ABB RAPID module: 711802ba.mod

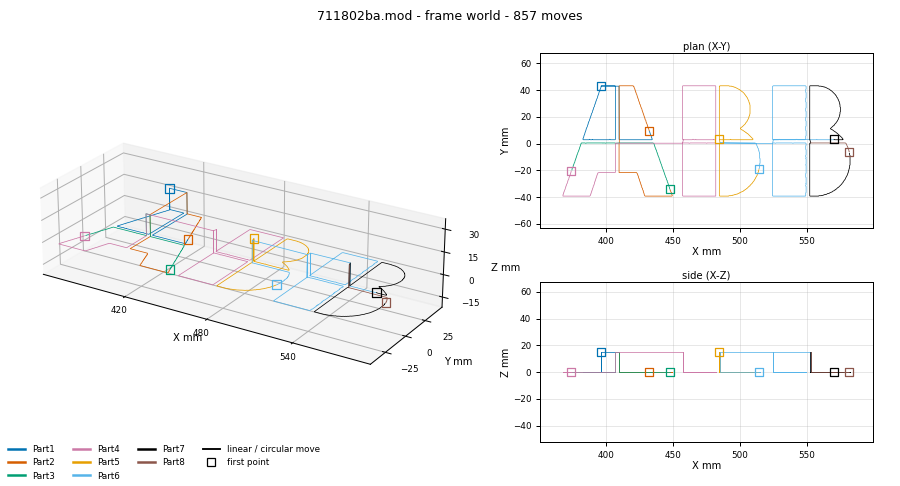
[picture p0: tool path of 711802ba.mod in frame world, 857 of 859 moves have a stored position in this frame; points joined in program order, loops and branches not executed]
MODULE ImageDraw
  ! Generated 2026-10-06 16:20 for ABB GoFa CRB 15000-5/0.95: 12 strokes
  PERS tooldata tPen:=[TRUE,[[0,0,120.0],[1,0,0,0]],[0.3,[0,0,60.0],[1,0,0,0],0,0,0]];
  PERS wobjdata wPaper:=[FALSE,TRUE,"",[[350,-90,0],[1,0,0,0]],[[0,0,0],[1,0,0,0]]];
  CONST robtarget pOrigin:=[[0,0,0],[0,1,0,0],[0,0,0,0],[9E9,9E9,9E9,9E9,9E9,9E9]];
  CONST jointtarget jHome:=[[0,0,0,0,30,0],[9E9,9E9,9E9,9E9,9E9,9E9]];
  CONST speeddata vDraw:=[40,100,5000,1000];
  CONST speeddata vApproach:=[20,100,5000,1000];
  CONST speeddata vTravel:=[200,200,5000,1000];

  PROC DrawImage()
    ConfL\Off;
    ConfJ\Off;
    MoveAbsJ jHome\NoEOffs,vTravel,fine,tPen;
    Part1;
    Part2;
    Part3;
    Part4;
    Part5;
    Part6;
    Part7;
    Part8;
    MoveAbsJ jHome\NoEOffs,vTravel,fine,tPen;
  ENDPROC

  PROC Part1()
    MoveL Offs(pOrigin,46.3,132.9,15.0),vTravel,z5,tPen\WObj:=wPaper;
    MoveL Offs(pOrigin,46.3,132.9,0.0),vApproach,fine,tPen\WObj:=wPaper;
    MoveL Offs(pOrigin,46.3,132.4,0.0),vDraw,z1,tPen\WObj:=wPaper;
    MoveL Offs(pOrigin,46.1,132.1,0.0),vDraw,z1,tPen\WObj:=wPaper;
    MoveL Offs(pOrigin,46.1,131.6,0.0),vDraw,z1,tPen\WObj:=wPaper;
    MoveL Offs(pOrigin,45.8,131.3,0.0),vDraw,z1,tPen\WObj:=wPaper;
    MoveL Offs(pOrigin,45.8,130.8,0.0),vDraw,z1,tPen\WObj:=wPaper;
    MoveL Offs(pOrigin,45.5,130.5,0.0),vDraw,z1,tPen\WObj:=wPaper;
    MoveL Offs(pOrigin,45.3,129.2,0.0),vDraw,z1,tPen\WObj:=wPaper;
    MoveL Offs(pOrigin,44.7,128.4,0.0),vDraw,z1,tPen\WObj:=wPaper;
    MoveL Offs(pOrigin,44.7,127.9,0.0),vDraw,z1,tPen\WObj:=wPaper;
    MoveL Offs(pOrigin,44.5,127.6,0.0),vDraw,z1,tPen\WObj:=wPaper;
    MoveL Offs(pOrigin,44.5,127.1,0.0),vDraw,z1,tPen\WObj:=wPaper;
    MoveL Offs(pOrigin,44.2,126.8,0.0),vDraw,z1,tPen\WObj:=wPaper;
    MoveL Offs(pOrigin,44.2,126.3,0.0),vDraw,z1,tPen\WObj:=wPaper;
    MoveL Offs(pOrigin,43.9,126.0,0.0),vDraw,z1,tPen\WObj:=wPaper;
    MoveL Offs(pOrigin,43.9,125.5,0.0),vDraw,z1,tPen\WObj:=wPaper;
    MoveL Offs(pOrigin,43.7,125.2,0.0),vDraw,z1,tPen\WObj:=wPaper;
    MoveL Offs(pOrigin,43.4,123.9,0.0),vDraw,z1,tPen\WObj:=wPaper;
    MoveL Offs(pOrigin,42.9,123.1,0.0),vDraw,z1,tPen\WObj:=wPaper;
    MoveL Offs(pOrigin,42.9,122.5,0.0),vDraw,z1,tPen\WObj:=wPaper;
    MoveL Offs(pOrigin,42.6,122.3,0.0),vDraw,z1,tPen\WObj:=wPaper;
    MoveL Offs(pOrigin,42.6,121.7,0.0),vDraw,z1,tPen\WObj:=wPaper;
    MoveL Offs(pOrigin,42.3,121.5,0.0),vDraw,z1,tPen\WObj:=wPaper;
    MoveL Offs(pOrigin,42.3,120.9,0.0),vDraw,z1,tPen\WObj:=wPaper;
    MoveL Offs(pOrigin,42.1,120.7,0.0),vDraw,z1,tPen\WObj:=wPaper;
    MoveL Offs(pOrigin,42.1,120.1,0.0),vDraw,z1,tPen\WObj:=wPaper;
    MoveL Offs(pOrigin,41.8,119.9,0.0),vDraw,z1,tPen\WObj:=wPaper;
    MoveL Offs(pOrigin,41.8,119.3,0.0),vDraw,z1,tPen\WObj:=wPaper;
    MoveL Offs(pOrigin,41.5,119.1,0.0),vDraw,z1,tPen\WObj:=wPaper;
    MoveL Offs(pOrigin,41.3,117.7,0.0),vDraw,z1,tPen\WObj:=wPaper;
    MoveL Offs(pOrigin,40.7,116.9,0.0),vDraw,z1,tPen\WObj:=wPaper;
    MoveL Offs(pOrigin,40.7,116.4,0.0),vDraw,z1,tPen\WObj:=wPaper;
    MoveL Offs(pOrigin,40.5,116.1,0.0),vDraw,z1,tPen\WObj:=wPaper;
    MoveL Offs(pOrigin,40.5,115.6,0.0),vDraw,z1,tPen\WObj:=wPaper;
    MoveL Offs(pOrigin,40.2,115.3,0.0),vDraw,z1,tPen\WObj:=wPaper;
    MoveL Offs(pOrigin,40.2,114.8,0.0),vDraw,z1,tPen\WObj:=wPaper;
    MoveL Offs(pOrigin,39.9,114.5,0.0),vDraw,z1,tPen\WObj:=wPaper;
    MoveL Offs(pOrigin,39.7,113.2,0.0),vDraw,z1,tPen\WObj:=wPaper;
    MoveL Offs(pOrigin,39.1,112.4,0.0),vDraw,z1,tPen\WObj:=wPaper;
    MoveL Offs(pOrigin,39.1,111.9,0.0),vDraw,z1,tPen\WObj:=wPaper;
    MoveL Offs(pOrigin,38.9,111.6,0.0),vDraw,z1,tPen\WObj:=wPaper;
    MoveL Offs(pOrigin,38.9,111.1,0.0),vDraw,z1,tPen\WObj:=wPaper;
    MoveL Offs(pOrigin,38.6,110.8,0.0),vDraw,z1,tPen\WObj:=wPaper;
    MoveL Offs(pOrigin,38.6,110.3,0.0),vDraw,z1,tPen\WObj:=wPaper;
    MoveL Offs(pOrigin,38.3,110.0,0.0),vDraw,z1,tPen\WObj:=wPaper;
    MoveL Offs(pOrigin,38.3,109.5,0.0),vDraw,z1,tPen\WObj:=wPaper;
    MoveL Offs(pOrigin,38.1,109.2,0.0),vDraw,z1,tPen\WObj:=wPaper;
    MoveL Offs(pOrigin,38.1,108.7,0.0),vDraw,z1,tPen\WObj:=wPaper;
    MoveL Offs(pOrigin,37.8,108.4,0.0),vDraw,z1,tPen\WObj:=wPaper;
    MoveL Offs(pOrigin,37.5,107.1,0.0),vDraw,z1,tPen\WObj:=wPaper;
    MoveL Offs(pOrigin,37.0,106.3,0.0),vDraw,z1,tPen\WObj:=wPaper;
    MoveL Offs(pOrigin,37.0,105.7,0.0),vDraw,z1,tPen\WObj:=wPaper;
    MoveL Offs(pOrigin,36.7,105.5,0.0),vDraw,z1,tPen\WObj:=wPaper;
    MoveL Offs(pOrigin,36.7,104.9,0.0),vDraw,z1,tPen\WObj:=wPaper;
    MoveL Offs(pOrigin,36.5,104.7,0.0),vDraw,z1,tPen\WObj:=wPaper;
    MoveL Offs(pOrigin,36.5,104.1,0.0),vDraw,z1,tPen\WObj:=wPaper;
    MoveL Offs(pOrigin,36.2,103.9,0.0),vDraw,z1,tPen\WObj:=wPaper;
    MoveL Offs(pOrigin,35.9,102.5,0.0),vDraw,z1,tPen\WObj:=wPaper;
    MoveL Offs(pOrigin,35.4,101.7,0.0),vDraw,z1,tPen\WObj:=wPaper;
    MoveL Offs(pOrigin,35.4,101.2,0.0),vDraw,z1,tPen\WObj:=wPaper;
    MoveL Offs(pOrigin,35.1,100.9,0.0),vDraw,z1,tPen\WObj:=wPaper;
    MoveL Offs(pOrigin,35.1,100.4,0.0),vDraw,z1,tPen\WObj:=wPaper;
    MoveL Offs(pOrigin,34.9,100.1,0.0),vDraw,z1,tPen\WObj:=wPaper;
    MoveL Offs(pOrigin,34.9,99.6,0.0),vDraw,z1,tPen\WObj:=wPaper;
    MoveL Offs(pOrigin,34.6,99.3,0.0),vDraw,z1,tPen\WObj:=wPaper;
    MoveL Offs(pOrigin,34.6,98.8,0.0),vDraw,z1,tPen\WObj:=wPaper;
    MoveL Offs(pOrigin,34.3,98.5,0.0),vDraw,z1,tPen\WObj:=wPaper;
    MoveL Offs(pOrigin,34.3,98.0,0.0),vDraw,z1,tPen\WObj:=wPaper;
    MoveL Offs(pOrigin,34.1,97.7,0.0),vDraw,z1,tPen\WObj:=wPaper;
    MoveL Offs(pOrigin,34.1,97.2,0.0),vDraw,z1,tPen\WObj:=wPaper;
    MoveL Offs(pOrigin,33.8,96.9,0.0),vDraw,z1,tPen\WObj:=wPaper;
    MoveL Offs(pOrigin,33.8,96.4,0.0),vDraw,z1,tPen\WObj:=wPaper;
    MoveL Offs(pOrigin,33.5,96.1,0.0),vDraw,z1,tPen\WObj:=wPaper;
    MoveL Offs(pOrigin,33.5,95.6,0.0),vDraw,z1,tPen\WObj:=wPaper;
    MoveL Offs(pOrigin,33.3,95.3,0.0),vDraw,z1,tPen\WObj:=wPaper;
    MoveL Offs(pOrigin,33.3,94.8,0.0),vDraw,z1,tPen\WObj:=wPaper;
    MoveL Offs(pOrigin,33.0,94.5,0.0),vDraw,z1,tPen\WObj:=wPaper;
    MoveL Offs(pOrigin,33.0,94.0,0.0),vDraw,z1,tPen\WObj:=wPaper;
    MoveL Offs(pOrigin,32.7,93.7,0.0),vDraw,z1,tPen\WObj:=wPaper;
    MoveL Offs(pOrigin,32.7,93.2,0.0),vDraw,z1,tPen\WObj:=wPaper;
    MoveL Offs(pOrigin,33.0,92.9,0.0),vDraw,z1,tPen\WObj:=wPaper;
    MoveL Offs(pOrigin,37.3,92.9,0.0),vDraw,z1,tPen\WObj:=wPaper;
    MoveL Offs(pOrigin,37.5,93.2,0.0),vDraw,z1,tPen\WObj:=wPaper;
    MoveL Offs(pOrigin,37.8,93.2,0.0),vDraw,z1,tPen\WObj:=wPaper;
    MoveL Offs(pOrigin,38.1,92.9,0.0),vDraw,z1,tPen\WObj:=wPaper;
    MoveL Offs(pOrigin,39.4,92.9,0.0),vDraw,z1,tPen\WObj:=wPaper;
    MoveL Offs(pOrigin,39.7,93.2,0.0),vDraw,z1,tPen\WObj:=wPaper;
    MoveL Offs(pOrigin,39.9,92.9,0.0),vDraw,z1,tPen\WObj:=wPaper;
    MoveL Offs(pOrigin,52.2,92.9,0.0),vDraw,z1,tPen\WObj:=wPaper;
    MoveL Offs(pOrigin,52.5,93.2,0.0),vDraw,z1,tPen\WObj:=wPaper;
    MoveL Offs(pOrigin,53.0,93.2,0.0),vDraw,z1,tPen\WObj:=wPaper;
    MoveL Offs(pOrigin,53.3,92.9,0.0),vDraw,z1,tPen\WObj:=wPaper;
    MoveL Offs(pOrigin,56.7,92.9,0.0),vDraw,z1,tPen\WObj:=wPaper;
    MoveL Offs(pOrigin,57.0,93.2,0.0),vDraw,z1,tPen\WObj:=wPaper;
    MoveL Offs(pOrigin,57.0,132.9,0.0),vDraw,z1,tPen\WObj:=wPaper;
    MoveL Offs(pOrigin,56.7,132.9,0.0),vDraw,z1,tPen\WObj:=wPaper;
    MoveL Offs(pOrigin,56.5,133.2,0.0),vDraw,z1,tPen\WObj:=wPaper;
    MoveL Offs(pOrigin,46.6,133.2,0.0),vDraw,z1,tPen\WObj:=wPaper;
    MoveL Offs(pOrigin,46.3,132.9,0.0),vDraw,fine,tPen\WObj:=wPaper;
    MoveL Offs(pOrigin,46.3,132.9,15.0),vApproach,z5,tPen\WObj:=wPaper;
    MoveL Offs(pOrigin,59.7,132.9,15.0),vTravel,z5,tPen\WObj:=wPaper;
    MoveL Offs(pOrigin,59.7,132.9,0.0),vApproach,fine,tPen\WObj:=wPaper;
    MoveL Offs(pOrigin,59.7,93.2,0.0),vDraw,z1,tPen\WObj:=wPaper;
    MoveL Offs(pOrigin,59.9,93.2,0.0),vDraw,z1,tPen\WObj:=wPaper;
    MoveL Offs(pOrigin,60.2,92.9,0.0),vDraw,z1,tPen\WObj:=wPaper;
    MoveL Offs(pOrigin,84.2,92.9,0.0),vDraw,z1,tPen\WObj:=wPaper;
    MoveL Offs(pOrigin,84.5,93.2,0.0),vDraw,z1,tPen\WObj:=wPaper;
    MoveL Offs(pOrigin,84.5,93.5,0.0),vDraw,z1,tPen\WObj:=wPaper;
    MoveL Offs(pOrigin,84.2,93.7,0.0),vDraw,z1,tPen\WObj:=wPaper;
    MoveL Offs(pOrigin,84.2,94.3,0.0),vDraw,z1,tPen\WObj:=wPaper;
    MoveL Offs(pOrigin,83.9,94.5,0.0),vDraw,z1,tPen\WObj:=wPaper;
    MoveL Offs(pOrigin,83.7,95.9,0.0),vDraw,z1,tPen\WObj:=wPaper;
    MoveL Offs(pOrigin,83.1,96.7,0.0),vDraw,z1,tPen\WObj:=wPaper;
    MoveL Offs(pOrigin,83.1,97.2,0.0),vDraw,z1,tPen\WObj:=wPaper;
    MoveL Offs(pOrigin,82.9,97.5,0.0),vDraw,z1,tPen\WObj:=wPaper;
    MoveL Offs(pOrigin,82.9,98.0,0.0),vDraw,z1,tPen\WObj:=wPaper;
    MoveL Offs(pOrigin,82.6,98.3,0.0),vDraw,z1,tPen\WObj:=wPaper;
    MoveL Offs(pOrigin,82.6,98.8,0.0),vDraw,z1,tPen\WObj:=wPaper;
    MoveL Offs(pOrigin,82.3,99.1,0.0),vDraw,z1,tPen\WObj:=wPaper;
  ENDPROC

  PROC Part2()
    MoveL Offs(pOrigin,82.3,99.6,0.0),vDraw,z1,tPen\WObj:=wPaper;
    MoveL Offs(pOrigin,82.1,99.9,0.0),vDraw,z1,tPen\WObj:=wPaper;
    MoveL Offs(pOrigin,81.8,101.2,0.0),vDraw,z1,tPen\WObj:=wPaper;
    MoveL Offs(pOrigin,81.5,101.5,0.0),vDraw,z1,tPen\WObj:=wPaper;
    MoveL Offs(pOrigin,81.5,101.7,0.0),vDraw,z1,tPen\WObj:=wPaper;
    MoveL Offs(pOrigin,81.3,102.0,0.0),vDraw,z1,tPen\WObj:=wPaper;
    MoveL Offs(pOrigin,81.3,102.5,0.0),vDraw,z1,tPen\WObj:=wPaper;
    MoveL Offs(pOrigin,81.0,102.8,0.0),vDraw,z1,tPen\WObj:=wPaper;
    MoveL Offs(pOrigin,81.0,103.6,0.0),vDraw,z1,tPen\WObj:=wPaper;
    MoveL Offs(pOrigin,80.7,103.9,0.0),vDraw,z1,tPen\WObj:=wPaper;
    MoveL Offs(pOrigin,80.7,104.4,0.0),vDraw,z1,tPen\WObj:=wPaper;
    MoveL Offs(pOrigin,80.2,105.2,0.0),vDraw,z1,tPen\WObj:=wPaper;
    MoveL Offs(pOrigin,80.2,105.7,0.0),vDraw,z1,tPen\WObj:=wPaper;
    MoveL Offs(pOrigin,79.9,106.0,0.0),vDraw,z1,tPen\WObj:=wPaper;
    MoveL Offs(pOrigin,79.7,107.3,0.0),vDraw,z1,tPen\WObj:=wPaper;
    MoveL Offs(pOrigin,79.1,108.1,0.0),vDraw,z1,tPen\WObj:=wPaper;
    MoveL Offs(pOrigin,79.1,108.7,0.0),vDraw,z1,tPen\WObj:=wPaper;
    MoveL Offs(pOrigin,78.9,108.9,0.0),vDraw,z1,tPen\WObj:=wPaper;
    MoveL Offs(pOrigin,78.9,109.5,0.0),vDraw,z1,tPen\WObj:=wPaper;
    MoveL Offs(pOrigin,78.6,109.7,0.0),vDraw,z1,tPen\WObj:=wPaper;
    MoveL Offs(pOrigin,78.6,110.3,0.0),vDraw,z1,tPen\WObj:=wPaper;
    MoveL Offs(pOrigin,78.3,110.5,0.0),vDraw,z1,tPen\WObj:=wPaper;
    MoveL Offs(pOrigin,78.3,111.1,0.0),vDraw,z1,tPen\WObj:=wPaper;
    MoveL Offs(pOrigin,78.1,111.3,0.0),vDraw,z1,tPen\WObj:=wPaper;
    MoveL Offs(pOrigin,78.1,111.9,0.0),vDraw,z1,tPen\WObj:=wPaper;
    MoveL Offs(pOrigin,77.8,112.1,0.0),vDraw,z1,tPen\WObj:=wPaper;
    MoveL Offs(pOrigin,77.8,112.7,0.0),vDraw,z1,tPen\WObj:=wPaper;
    MoveL Offs(pOrigin,77.5,112.9,0.0),vDraw,z1,tPen\WObj:=wPaper;
    MoveL Offs(pOrigin,77.5,113.5,0.0),vDraw,z1,tPen\WObj:=wPaper;
    MoveL Offs(pOrigin,77.3,113.7,0.0),vDraw,z1,tPen\WObj:=wPaper;
    MoveL Offs(pOrigin,77.3,114.3,0.0),vDraw,z1,tPen\WObj:=wPaper;
    MoveL Offs(pOrigin,77.0,114.5,0.0),vDraw,z1,tPen\WObj:=wPaper;
    MoveL Offs(pOrigin,76.7,115.9,0.0),vDraw,z1,tPen\WObj:=wPaper;
    MoveL Offs(pOrigin,76.2,116.7,0.0),vDraw,z1,tPen\WObj:=wPaper;
    MoveL Offs(pOrigin,76.2,117.2,0.0),vDraw,z1,tPen\WObj:=wPaper;
    MoveL Offs(pOrigin,75.9,117.5,0.0),vDraw,z1,tPen\WObj:=wPaper;
    MoveL Offs(pOrigin,75.7,118.8,0.0),vDraw,z1,tPen\WObj:=wPaper;
    MoveL Offs(pOrigin,75.1,119.6,0.0),vDraw,z1,tPen\WObj:=wPaper;
    MoveL Offs(pOrigin,75.1,120.1,0.0),vDraw,z1,tPen\WObj:=wPaper;
    MoveL Offs(pOrigin,74.9,120.4,0.0),vDraw,z1,tPen\WObj:=wPaper;
    MoveL Offs(pOrigin,74.9,120.9,0.0),vDraw,z1,tPen\WObj:=wPaper;
    MoveL Offs(pOrigin,74.6,121.2,0.0),vDraw,z1,tPen\WObj:=wPaper;
    MoveL Offs(pOrigin,74.6,121.7,0.0),vDraw,z1,tPen\WObj:=wPaper;
    MoveL Offs(pOrigin,74.3,122.0,0.0),vDraw,z1,tPen\WObj:=wPaper;
    MoveL Offs(pOrigin,74.3,122.5,0.0),vDraw,z1,tPen\WObj:=wPaper;
    MoveL Offs(pOrigin,74.1,122.8,0.0),vDraw,z1,tPen\WObj:=wPaper;
    MoveL Offs(pOrigin,74.1,123.3,0.0),vDraw,z1,tPen\WObj:=wPaper;
    MoveL Offs(pOrigin,73.8,123.6,0.0),vDraw,z1,tPen\WObj:=wPaper;
    MoveL Offs(pOrigin,73.8,124.1,0.0),vDraw,z1,tPen\WObj:=wPaper;
    MoveL Offs(pOrigin,73.5,124.4,0.0),vDraw,z1,tPen\WObj:=wPaper;
    MoveL Offs(pOrigin,73.5,124.9,0.0),vDraw,z1,tPen\WObj:=wPaper;
    MoveL Offs(pOrigin,73.3,125.2,0.0),vDraw,z1,tPen\WObj:=wPaper;
    MoveL Offs(pOrigin,73.0,126.5,0.0),vDraw,z1,tPen\WObj:=wPaper;
    MoveL Offs(pOrigin,72.5,127.3,0.0),vDraw,z1,tPen\WObj:=wPaper;
    MoveL Offs(pOrigin,72.5,127.9,0.0),vDraw,z1,tPen\WObj:=wPaper;
    MoveL Offs(pOrigin,72.2,128.1,0.0),vDraw,z1,tPen\WObj:=wPaper;
    MoveL Offs(pOrigin,72.2,128.7,0.0),vDraw,z1,tPen\WObj:=wPaper;
    MoveL Offs(pOrigin,71.9,128.9,0.0),vDraw,z1,tPen\WObj:=wPaper;
    MoveL Offs(pOrigin,71.9,129.5,0.0),vDraw,z1,tPen\WObj:=wPaper;
    MoveL Offs(pOrigin,71.7,129.7,0.0),vDraw,z1,tPen\WObj:=wPaper;
    MoveL Offs(pOrigin,71.7,130.3,0.0),vDraw,z1,tPen\WObj:=wPaper;
    MoveL Offs(pOrigin,71.4,130.5,0.0),vDraw,z1,tPen\WObj:=wPaper;
    MoveL Offs(pOrigin,71.4,131.1,0.0),vDraw,z1,tPen\WObj:=wPaper;
    MoveL Offs(pOrigin,70.9,131.9,0.0),vDraw,z1,tPen\WObj:=wPaper;
    MoveL Offs(pOrigin,70.9,132.4,0.0),vDraw,z1,tPen\WObj:=wPaper;
    MoveL Offs(pOrigin,70.6,132.7,0.0),vDraw,z1,tPen\WObj:=wPaper;
    MoveL Offs(pOrigin,70.6,132.9,0.0),vDraw,z1,tPen\WObj:=wPaper;
    MoveL Offs(pOrigin,70.3,132.9,0.0),vDraw,z1,tPen\WObj:=wPaper;
    MoveL Offs(pOrigin,70.1,133.2,0.0),vDraw,z1,tPen\WObj:=wPaper;
    MoveL Offs(pOrigin,59.9,133.2,0.0),vDraw,z1,tPen\WObj:=wPaper;
    MoveL Offs(pOrigin,59.7,132.9,0.0),vDraw,fine,tPen\WObj:=wPaper;
    MoveL Offs(pOrigin,59.7,132.9,15.0),vApproach,z5,tPen\WObj:=wPaper;
    MoveL Offs(pOrigin,59.9,90.5,15.0),vTravel,z5,tPen\WObj:=wPaper;
    MoveL Offs(pOrigin,59.9,90.5,0.0),vApproach,fine,tPen\WObj:=wPaper;
    MoveL Offs(pOrigin,59.7,90.3,0.0),vDraw,z1,tPen\WObj:=wPaper;
    MoveL Offs(pOrigin,59.7,68.4,0.0),vDraw,z1,tPen\WObj:=wPaper;
    MoveL Offs(pOrigin,72.7,68.4,0.0),vDraw,z1,tPen\WObj:=wPaper;
    MoveL Offs(pOrigin,73.5,67.3,0.0),vDraw,z1,tPen\WObj:=wPaper;
    MoveL Offs(pOrigin,73.5,66.8,0.0),vDraw,z1,tPen\WObj:=wPaper;
    MoveL Offs(pOrigin,73.8,66.5,0.0),vDraw,z1,tPen\WObj:=wPaper;
    MoveL Offs(pOrigin,73.8,66.0,0.0),vDraw,z1,tPen\WObj:=wPaper;
    MoveL Offs(pOrigin,74.1,65.7,0.0),vDraw,z1,tPen\WObj:=wPaper;
    MoveL Offs(pOrigin,74.1,65.2,0.0),vDraw,z1,tPen\WObj:=wPaper;
    MoveL Offs(pOrigin,74.3,64.9,0.0),vDraw,z1,tPen\WObj:=wPaper;
    MoveL Offs(pOrigin,74.3,64.4,0.0),vDraw,z1,tPen\WObj:=wPaper;
    MoveL Offs(pOrigin,74.6,64.1,0.0),vDraw,z1,tPen\WObj:=wPaper;
    MoveL Offs(pOrigin,74.6,63.6,0.0),vDraw,z1,tPen\WObj:=wPaper;
    MoveL Offs(pOrigin,74.9,63.3,0.0),vDraw,z1,tPen\WObj:=wPaper;
    MoveL Offs(pOrigin,74.9,62.8,0.0),vDraw,z1,tPen\WObj:=wPaper;
    MoveL Offs(pOrigin,75.1,62.5,0.0),vDraw,z1,tPen\WObj:=wPaper;
    MoveL Offs(pOrigin,75.1,62.0,0.0),vDraw,z1,tPen\WObj:=wPaper;
    MoveL Offs(pOrigin,75.4,61.7,0.0),vDraw,z1,tPen\WObj:=wPaper;
    MoveL Offs(pOrigin,75.4,61.2,0.0),vDraw,z1,tPen\WObj:=wPaper;
    MoveL Offs(pOrigin,75.7,60.9,0.0),vDraw,z1,tPen\WObj:=wPaper;
    MoveL Offs(pOrigin,75.7,60.4,0.0),vDraw,z1,tPen\WObj:=wPaper;
    MoveL Offs(pOrigin,75.9,60.1,0.0),vDraw,z1,tPen\WObj:=wPaper;
    MoveL Offs(pOrigin,75.9,59.6,0.0),vDraw,z1,tPen\WObj:=wPaper;
    MoveL Offs(pOrigin,76.2,59.3,0.0),vDraw,z1,tPen\WObj:=wPaper;
    MoveL Offs(pOrigin,76.2,58.8,0.0),vDraw,z1,tPen\WObj:=wPaper;
    MoveL Offs(pOrigin,76.5,58.5,0.0),vDraw,z1,tPen\WObj:=wPaper;
    MoveL Offs(pOrigin,76.7,57.2,0.0),vDraw,z1,tPen\WObj:=wPaper;
    MoveL Offs(pOrigin,77.3,56.4,0.0),vDraw,z1,tPen\WObj:=wPaper;
    MoveL Offs(pOrigin,77.3,55.6,0.0),vDraw,z1,tPen\WObj:=wPaper;
    MoveL Offs(pOrigin,77.8,54.8,0.0),vDraw,z1,tPen\WObj:=wPaper;
    MoveL Offs(pOrigin,77.8,54.0,0.0),vDraw,z1,tPen\WObj:=wPaper;
    MoveL Offs(pOrigin,78.1,53.7,0.0),vDraw,z1,tPen\WObj:=wPaper;
    MoveL Offs(pOrigin,78.1,53.2,0.0),vDraw,z1,tPen\WObj:=wPaper;
    MoveL Offs(pOrigin,78.3,52.9,0.0),vDraw,z1,tPen\WObj:=wPaper;
    MoveL Offs(pOrigin,78.6,51.6,0.0),vDraw,z1,tPen\WObj:=wPaper;
    MoveL Offs(pOrigin,79.1,50.8,0.0),vDraw,z1,tPen\WObj:=wPaper;
    MoveL Offs(pOrigin,99.1,50.8,0.0),vDraw,z1,tPen\WObj:=wPaper;
    MoveL Offs(pOrigin,99.4,51.1,0.0),vDraw,z1,tPen\WObj:=wPaper;
    MoveL Offs(pOrigin,99.4,51.6,0.0),vDraw,z1,tPen\WObj:=wPaper;
    MoveL Offs(pOrigin,99.1,51.9,0.0),vDraw,z1,tPen\WObj:=wPaper;
    MoveL Offs(pOrigin,98.9,53.2,0.0),vDraw,z1,tPen\WObj:=wPaper;
    MoveL Offs(pOrigin,98.6,53.5,0.0),vDraw,z1,tPen\WObj:=wPaper;
    MoveL Offs(pOrigin,98.6,53.7,0.0),vDraw,z1,tPen\WObj:=wPaper;
    MoveL Offs(pOrigin,98.3,54.0,0.0),vDraw,z1,tPen\WObj:=wPaper;
    MoveL Offs(pOrigin,98.3,54.5,0.0),vDraw,z1,tPen\WObj:=wPaper;
    MoveL Offs(pOrigin,97.8,55.3,0.0),vDraw,z1,tPen\WObj:=wPaper;
  ENDPROC

  PROC Part3()
    MoveL Offs(pOrigin,97.8,55.9,0.0),vDraw,z1,tPen\WObj:=wPaper;
    MoveL Offs(pOrigin,97.5,56.1,0.0),vDraw,z1,tPen\WObj:=wPaper;
    MoveL Offs(pOrigin,97.5,56.7,0.0),vDraw,z1,tPen\WObj:=wPaper;
    MoveL Offs(pOrigin,97.3,56.9,0.0),vDraw,z1,tPen\WObj:=wPaper;
    MoveL Offs(pOrigin,97.3,57.5,0.0),vDraw,z1,tPen\WObj:=wPaper;
    MoveL Offs(pOrigin,97.0,57.7,0.0),vDraw,z1,tPen\WObj:=wPaper;
    MoveL Offs(pOrigin,97.0,58.3,0.0),vDraw,z1,tPen\WObj:=wPaper;
    MoveL Offs(pOrigin,96.7,58.5,0.0),vDraw,z1,tPen\WObj:=wPaper;
    MoveL Offs(pOrigin,96.7,59.1,0.0),vDraw,z1,tPen\WObj:=wPaper;
    MoveL Offs(pOrigin,96.5,59.3,0.0),vDraw,z1,tPen\WObj:=wPaper;
    MoveL Offs(pOrigin,96.2,60.7,0.0),vDraw,z1,tPen\WObj:=wPaper;
    MoveL Offs(pOrigin,95.7,61.5,0.0),vDraw,z1,tPen\WObj:=wPaper;
    MoveL Offs(pOrigin,95.7,62.3,0.0),vDraw,z1,tPen\WObj:=wPaper;
    MoveL Offs(pOrigin,95.1,63.1,0.0),vDraw,z1,tPen\WObj:=wPaper;
    MoveL Offs(pOrigin,94.9,64.4,0.0),vDraw,z1,tPen\WObj:=wPaper;
    MoveL Offs(pOrigin,94.3,65.2,0.0),vDraw,z1,tPen\WObj:=wPaper;
    MoveL Offs(pOrigin,94.3,65.7,0.0),vDraw,z1,tPen\WObj:=wPaper;
    MoveL Offs(pOrigin,94.1,66.0,0.0),vDraw,z1,tPen\WObj:=wPaper;
    MoveL Offs(pOrigin,94.1,66.5,0.0),vDraw,z1,tPen\WObj:=wPaper;
    MoveL Offs(pOrigin,93.8,66.8,0.0),vDraw,z1,tPen\WObj:=wPaper;
    MoveL Offs(pOrigin,93.8,67.3,0.0),vDraw,z1,tPen\WObj:=wPaper;
    MoveL Offs(pOrigin,93.5,67.6,0.0),vDraw,z1,tPen\WObj:=wPaper;
    MoveL Offs(pOrigin,93.5,68.1,0.0),vDraw,z1,tPen\WObj:=wPaper;
    MoveL Offs(pOrigin,93.3,68.4,0.0),vDraw,z1,tPen\WObj:=wPaper;
    MoveL Offs(pOrigin,93.3,68.9,0.0),vDraw,z1,tPen\WObj:=wPaper;
    MoveL Offs(pOrigin,93.0,69.2,0.0),vDraw,z1,tPen\WObj:=wPaper;
    MoveL Offs(pOrigin,92.7,70.5,0.0),vDraw,z1,tPen\WObj:=wPaper;
    MoveL Offs(pOrigin,92.2,71.3,0.0),vDraw,z1,tPen\WObj:=wPaper;
    MoveL Offs(pOrigin,92.2,71.9,0.0),vDraw,z1,tPen\WObj:=wPaper;
    MoveL Offs(pOrigin,91.9,72.1,0.0),vDraw,z1,tPen\WObj:=wPaper;
    MoveL Offs(pOrigin,91.9,72.7,0.0),vDraw,z1,tPen\WObj:=wPaper;
    MoveL Offs(pOrigin,91.7,72.9,0.0),vDraw,z1,tPen\WObj:=wPaper;
    MoveL Offs(pOrigin,91.4,74.3,0.0),vDraw,z1,tPen\WObj:=wPaper;
    MoveL Offs(pOrigin,90.9,75.1,0.0),vDraw,z1,tPen\WObj:=wPaper;
    MoveL Offs(pOrigin,90.9,75.6,0.0),vDraw,z1,tPen\WObj:=wPaper;
    MoveL Offs(pOrigin,90.6,75.9,0.0),vDraw,z1,tPen\WObj:=wPaper;
    MoveL Offs(pOrigin,90.6,76.4,0.0),vDraw,z1,tPen\WObj:=wPaper;
    MoveL Offs(pOrigin,90.3,76.7,0.0),vDraw,z1,tPen\WObj:=wPaper;
    MoveL Offs(pOrigin,90.3,77.2,0.0),vDraw,z1,tPen\WObj:=wPaper;
    MoveL Offs(pOrigin,90.1,77.5,0.0),vDraw,z1,tPen\WObj:=wPaper;
    MoveL Offs(pOrigin,90.1,78.0,0.0),vDraw,z1,tPen\WObj:=wPaper;
    MoveL Offs(pOrigin,89.8,78.3,0.0),vDraw,z1,tPen\WObj:=wPaper;
    MoveL Offs(pOrigin,89.5,79.6,0.0),vDraw,z1,tPen\WObj:=wPaper;
    MoveL Offs(pOrigin,89.0,80.4,0.0),vDraw,z1,tPen\WObj:=wPaper;
    MoveL Offs(pOrigin,89.0,80.9,0.0),vDraw,z1,tPen\WObj:=wPaper;
    MoveL Offs(pOrigin,88.7,81.2,0.0),vDraw,z1,tPen\WObj:=wPaper;
    MoveL Offs(pOrigin,88.7,81.7,0.0),vDraw,z1,tPen\WObj:=wPaper;
    MoveL Offs(pOrigin,88.5,82.0,0.0),vDraw,z1,tPen\WObj:=wPaper;
    MoveL Offs(pOrigin,88.5,82.5,0.0),vDraw,z1,tPen\WObj:=wPaper;
    MoveL Offs(pOrigin,88.2,82.8,0.0),vDraw,z1,tPen\WObj:=wPaper;
    MoveL Offs(pOrigin,88.2,83.3,0.0),vDraw,z1,tPen\WObj:=wPaper;
    MoveL Offs(pOrigin,87.9,83.6,0.0),vDraw,z1,tPen\WObj:=wPaper;
    MoveL Offs(pOrigin,87.7,84.9,0.0),vDraw,z1,tPen\WObj:=wPaper;
    MoveL Offs(pOrigin,87.4,85.2,0.0),vDraw,z1,tPen\WObj:=wPaper;
    MoveL Offs(pOrigin,87.4,85.5,0.0),vDraw,z1,tPen\WObj:=wPaper;
    MoveL Offs(pOrigin,87.1,85.7,0.0),vDraw,z1,tPen\WObj:=wPaper;
    MoveL Offs(pOrigin,87.1,86.3,0.0),vDraw,z1,tPen\WObj:=wPaper;
    MoveL Offs(pOrigin,86.6,87.1,0.0),vDraw,z1,tPen\WObj:=wPaper;
    MoveL Offs(pOrigin,86.6,87.6,0.0),vDraw,z1,tPen\WObj:=wPaper;
    MoveL Offs(pOrigin,86.3,87.9,0.0),vDraw,z1,tPen\WObj:=wPaper;
    MoveL Offs(pOrigin,86.3,88.4,0.0),vDraw,z1,tPen\WObj:=wPaper;
    MoveL Offs(pOrigin,86.1,88.7,0.0),vDraw,z1,tPen\WObj:=wPaper;
    MoveL Offs(pOrigin,85.8,90.0,0.0),vDraw,z1,tPen\WObj:=wPaper;
    MoveL Offs(pOrigin,85.0,90.5,0.0),vDraw,z1,tPen\WObj:=wPaper;
    MoveL Offs(pOrigin,59.9,90.5,0.0),vDraw,fine,tPen\WObj:=wPaper;
    MoveL Offs(pOrigin,59.9,90.5,15.0),vApproach,z5,tPen\WObj:=wPaper;
    MoveL Offs(pOrigin,57.0,90.3,15.0),vTravel,z5,tPen\WObj:=wPaper;
    MoveL Offs(pOrigin,57.0,90.3,0.0),vApproach,fine,tPen\WObj:=wPaper;
    MoveL Offs(pOrigin,56.7,90.3,0.0),vDraw,z1,tPen\WObj:=wPaper;
    MoveL Offs(pOrigin,56.5,90.5,0.0),vDraw,z1,tPen\WObj:=wPaper;
    MoveL Offs(pOrigin,49.8,90.5,0.0),vDraw,z1,tPen\WObj:=wPaper;
    MoveL Offs(pOrigin,49.5,90.3,0.0),vDraw,z1,tPen\WObj:=wPaper;
    MoveL Offs(pOrigin,49.3,90.3,0.0),vDraw,z1,tPen\WObj:=wPaper;
    MoveL Offs(pOrigin,49.0,90.5,0.0),vDraw,z1,tPen\WObj:=wPaper;
    MoveL Offs(pOrigin,47.9,90.5,0.0),vDraw,z1,tPen\WObj:=wPaper;
    MoveL Offs(pOrigin,47.7,90.3,0.0),vDraw,z1,tPen\WObj:=wPaper;
    MoveL Offs(pOrigin,47.4,90.5,0.0),vDraw,z1,tPen\WObj:=wPaper;
    MoveL Offs(pOrigin,35.4,90.5,0.0),vDraw,z1,tPen\WObj:=wPaper;
    MoveL Offs(pOrigin,35.1,90.3,0.0),vDraw,z1,tPen\WObj:=wPaper;
    MoveL Offs(pOrigin,34.6,90.3,0.0),vDraw,z1,tPen\WObj:=wPaper;
    MoveL Offs(pOrigin,34.3,90.5,0.0),vDraw,z1,tPen\WObj:=wPaper;
    MoveL Offs(pOrigin,31.7,90.5,0.0),vDraw,z1,tPen\WObj:=wPaper;
    MoveL Offs(pOrigin,31.4,90.3,0.0),vDraw,z1,tPen\WObj:=wPaper;
    MoveL Offs(pOrigin,31.4,90.0,0.0),vDraw,z1,tPen\WObj:=wPaper;
    MoveL Offs(pOrigin,31.1,89.7,0.0),vDraw,z1,tPen\WObj:=wPaper;
    MoveL Offs(pOrigin,31.1,89.2,0.0),vDraw,z1,tPen\WObj:=wPaper;
    MoveL Offs(pOrigin,30.9,88.9,0.0),vDraw,z1,tPen\WObj:=wPaper;
    MoveL Offs(pOrigin,30.9,88.4,0.0),vDraw,z1,tPen\WObj:=wPaper;
    MoveL Offs(pOrigin,30.6,88.1,0.0),vDraw,z1,tPen\WObj:=wPaper;
    MoveL Offs(pOrigin,30.6,87.6,0.0),vDraw,z1,tPen\WObj:=wPaper;
    MoveL Offs(pOrigin,30.3,87.3,0.0),vDraw,z1,tPen\WObj:=wPaper;
    MoveL Offs(pOrigin,30.3,86.8,0.0),vDraw,z1,tPen\WObj:=wPaper;
    MoveL Offs(pOrigin,30.1,86.5,0.0),vDraw,z1,tPen\WObj:=wPaper;
    MoveL Offs(pOrigin,30.1,86.0,0.0),vDraw,z1,tPen\WObj:=wPaper;
    MoveL Offs(pOrigin,29.8,85.7,0.0),vDraw,z1,tPen\WObj:=wPaper;
    MoveL Offs(pOrigin,29.8,85.2,0.0),vDraw,z1,tPen\WObj:=wPaper;
    MoveL Offs(pOrigin,29.3,84.4,0.0),vDraw,z1,tPen\WObj:=wPaper;
    MoveL Offs(pOrigin,29.3,83.9,0.0),vDraw,z1,tPen\WObj:=wPaper;
    MoveL Offs(pOrigin,29.0,83.6,0.0),vDraw,z1,tPen\WObj:=wPaper;
    MoveL Offs(pOrigin,28.7,82.3,0.0),vDraw,z1,tPen\WObj:=wPaper;
    MoveL Offs(pOrigin,28.2,81.5,0.0),vDraw,z1,tPen\WObj:=wPaper;
    MoveL Offs(pOrigin,28.2,80.9,0.0),vDraw,z1,tPen\WObj:=wPaper;
    MoveL Offs(pOrigin,27.9,80.7,0.0),vDraw,z1,tPen\WObj:=wPaper;
    MoveL Offs(pOrigin,27.9,80.1,0.0),vDraw,z1,tPen\WObj:=wPaper;
    MoveL Offs(pOrigin,27.7,79.9,0.0),vDraw,z1,tPen\WObj:=wPaper;
    MoveL Offs(pOrigin,27.7,79.3,0.0),vDraw,z1,tPen\WObj:=wPaper;
    MoveL Offs(pOrigin,27.4,79.1,0.0),vDraw,z1,tPen\WObj:=wPaper;
    MoveL Offs(pOrigin,27.4,78.5,0.0),vDraw,z1,tPen\WObj:=wPaper;
    MoveL Offs(pOrigin,27.1,78.3,0.0),vDraw,z1,tPen\WObj:=wPaper;
    MoveL Offs(pOrigin,27.1,77.7,0.0),vDraw,z1,tPen\WObj:=wPaper;
    MoveL Offs(pOrigin,26.9,77.5,0.0),vDraw,z1,tPen\WObj:=wPaper;
    MoveL Offs(pOrigin,26.6,76.1,0.0),vDraw,z1,tPen\WObj:=wPaper;
    MoveL Offs(pOrigin,26.1,75.3,0.0),vDraw,z1,tPen\WObj:=wPaper;
    MoveL Offs(pOrigin,26.1,74.8,0.0),vDraw,z1,tPen\WObj:=wPaper;
    MoveL Offs(pOrigin,25.8,74.5,0.0),vDraw,z1,tPen\WObj:=wPaper;
    MoveL Offs(pOrigin,25.8,74.0,0.0),vDraw,z1,tPen\WObj:=wPaper;
    MoveL Offs(pOrigin,25.5,73.7,0.0),vDraw,z1,tPen\WObj:=wPaper;
    MoveL Offs(pOrigin,25.3,72.4,0.0),vDraw,z1,tPen\WObj:=wPaper;
    MoveL Offs(pOrigin,24.7,71.6,0.0),vDraw,z1,tPen\WObj:=wPaper;
    MoveL Offs(pOrigin,24.5,70.3,0.0),vDraw,z1,tPen\WObj:=wPaper;
  ENDPROC

  PROC Part4()
    MoveL Offs(pOrigin,23.9,69.5,0.0),vDraw,z1,tPen\WObj:=wPaper;
    MoveL Offs(pOrigin,23.9,68.9,0.0),vDraw,z1,tPen\WObj:=wPaper;
    MoveL Offs(pOrigin,23.7,68.7,0.0),vDraw,z1,tPen\WObj:=wPaper;
    MoveL Offs(pOrigin,23.7,68.1,0.0),vDraw,z1,tPen\WObj:=wPaper;
    MoveL Offs(pOrigin,23.4,67.9,0.0),vDraw,z1,tPen\WObj:=wPaper;
    MoveL Offs(pOrigin,23.4,67.1,0.0),vDraw,z1,tPen\WObj:=wPaper;
    MoveL Offs(pOrigin,22.9,66.3,0.0),vDraw,z1,tPen\WObj:=wPaper;
    MoveL Offs(pOrigin,22.9,65.7,0.0),vDraw,z1,tPen\WObj:=wPaper;
    MoveL Offs(pOrigin,22.6,65.5,0.0),vDraw,z1,tPen\WObj:=wPaper;
    MoveL Offs(pOrigin,22.6,64.9,0.0),vDraw,z1,tPen\WObj:=wPaper;
    MoveL Offs(pOrigin,22.3,64.7,0.0),vDraw,z1,tPen\WObj:=wPaper;
    MoveL Offs(pOrigin,22.1,63.3,0.0),vDraw,z1,tPen\WObj:=wPaper;
    MoveL Offs(pOrigin,21.5,62.5,0.0),vDraw,z1,tPen\WObj:=wPaper;
    MoveL Offs(pOrigin,21.5,62.0,0.0),vDraw,z1,tPen\WObj:=wPaper;
    MoveL Offs(pOrigin,21.3,61.7,0.0),vDraw,z1,tPen\WObj:=wPaper;
    MoveL Offs(pOrigin,21.0,60.4,0.0),vDraw,z1,tPen\WObj:=wPaper;
    MoveL Offs(pOrigin,20.5,59.6,0.0),vDraw,z1,tPen\WObj:=wPaper;
    MoveL Offs(pOrigin,20.5,59.1,0.0),vDraw,z1,tPen\WObj:=wPaper;
    MoveL Offs(pOrigin,20.2,58.8,0.0),vDraw,z1,tPen\WObj:=wPaper;
    MoveL Offs(pOrigin,20.2,58.3,0.0),vDraw,z1,tPen\WObj:=wPaper;
    MoveL Offs(pOrigin,19.9,58.0,0.0),vDraw,z1,tPen\WObj:=wPaper;
    MoveL Offs(pOrigin,19.9,57.5,0.0),vDraw,z1,tPen\WObj:=wPaper;
    MoveL Offs(pOrigin,19.7,57.2,0.0),vDraw,z1,tPen\WObj:=wPaper;
    MoveL Offs(pOrigin,19.4,55.9,0.0),vDraw,z1,tPen\WObj:=wPaper;
    MoveL Offs(pOrigin,18.9,55.1,0.0),vDraw,z1,tPen\WObj:=wPaper;
    MoveL Offs(pOrigin,18.9,54.5,0.0),vDraw,z1,tPen\WObj:=wPaper;
    MoveL Offs(pOrigin,18.6,54.3,0.0),vDraw,z1,tPen\WObj:=wPaper;
    MoveL Offs(pOrigin,18.6,53.7,0.0),vDraw,z1,tPen\WObj:=wPaper;
    MoveL Offs(pOrigin,18.3,53.5,0.0),vDraw,z1,tPen\WObj:=wPaper;
    MoveL Offs(pOrigin,18.3,52.9,0.0),vDraw,z1,tPen\WObj:=wPaper;
    MoveL Offs(pOrigin,18.1,52.7,0.0),vDraw,z1,tPen\WObj:=wPaper;
    MoveL Offs(pOrigin,18.1,52.1,0.0),vDraw,z1,tPen\WObj:=wPaper;
    MoveL Offs(pOrigin,17.8,51.9,0.0),vDraw,z1,tPen\WObj:=wPaper;
    MoveL Offs(pOrigin,17.8,50.8,0.0),vDraw,z1,tPen\WObj:=wPaper;
    MoveL Offs(pOrigin,37.8,50.8,0.0),vDraw,z1,tPen\WObj:=wPaper;
    MoveL Offs(pOrigin,38.3,51.3,0.0),vDraw,z1,tPen\WObj:=wPaper;
    MoveL Offs(pOrigin,38.3,51.9,0.0),vDraw,z1,tPen\WObj:=wPaper;
    MoveL Offs(pOrigin,38.6,52.1,0.0),vDraw,z1,tPen\WObj:=wPaper;
    MoveL Offs(pOrigin,38.6,52.7,0.0),vDraw,z1,tPen\WObj:=wPaper;
    MoveL Offs(pOrigin,38.9,52.9,0.0),vDraw,z1,tPen\WObj:=wPaper;
    MoveL Offs(pOrigin,38.9,53.5,0.0),vDraw,z1,tPen\WObj:=wPaper;
    MoveL Offs(pOrigin,39.1,53.7,0.0),vDraw,z1,tPen\WObj:=wPaper;
    MoveL Offs(pOrigin,39.1,54.3,0.0),vDraw,z1,tPen\WObj:=wPaper;
    MoveL Offs(pOrigin,39.4,54.5,0.0),vDraw,z1,tPen\WObj:=wPaper;
    MoveL Offs(pOrigin,39.4,55.1,0.0),vDraw,z1,tPen\WObj:=wPaper;
    MoveL Offs(pOrigin,39.7,55.3,0.0),vDraw,z1,tPen\WObj:=wPaper;
    MoveL Offs(pOrigin,39.7,55.9,0.0),vDraw,z1,tPen\WObj:=wPaper;
    MoveL Offs(pOrigin,39.9,56.1,0.0),vDraw,z1,tPen\WObj:=wPaper;
    MoveL Offs(pOrigin,39.9,56.7,0.0),vDraw,z1,tPen\WObj:=wPaper;
    MoveL Offs(pOrigin,40.2,56.9,0.0),vDraw,z1,tPen\WObj:=wPaper;
    MoveL Offs(pOrigin,40.5,58.3,0.0),vDraw,z1,tPen\WObj:=wPaper;
    MoveL Offs(pOrigin,41.0,59.1,0.0),vDraw,z1,tPen\WObj:=wPaper;
    MoveL Offs(pOrigin,41.0,59.6,0.0),vDraw,z1,tPen\WObj:=wPaper;
    MoveL Offs(pOrigin,41.3,59.9,0.0),vDraw,z1,tPen\WObj:=wPaper;
    MoveL Offs(pOrigin,41.3,60.7,0.0),vDraw,z1,tPen\WObj:=wPaper;
    MoveL Offs(pOrigin,41.5,60.9,0.0),vDraw,z1,tPen\WObj:=wPaper;
    MoveL Offs(pOrigin,41.5,61.5,0.0),vDraw,z1,tPen\WObj:=wPaper;
    MoveL Offs(pOrigin,41.8,61.7,0.0),vDraw,z1,tPen\WObj:=wPaper;
    MoveL Offs(pOrigin,41.8,62.3,0.0),vDraw,z1,tPen\WObj:=wPaper;
    MoveL Offs(pOrigin,42.1,62.5,0.0),vDraw,z1,tPen\WObj:=wPaper;
    MoveL Offs(pOrigin,42.1,63.1,0.0),vDraw,z1,tPen\WObj:=wPaper;
    MoveL Offs(pOrigin,42.3,63.3,0.0),vDraw,z1,tPen\WObj:=wPaper;
    MoveL Offs(pOrigin,42.3,63.9,0.0),vDraw,z1,tPen\WObj:=wPaper;
    MoveL Offs(pOrigin,42.6,64.1,0.0),vDraw,z1,tPen\WObj:=wPaper;
    MoveL Offs(pOrigin,42.6,64.7,0.0),vDraw,z1,tPen\WObj:=wPaper;
    MoveL Offs(pOrigin,42.9,64.9,0.0),vDraw,z1,tPen\WObj:=wPaper;
    MoveL Offs(pOrigin,42.9,65.5,0.0),vDraw,z1,tPen\WObj:=wPaper;
    MoveL Offs(pOrigin,43.1,65.7,0.0),vDraw,z1,tPen\WObj:=wPaper;
    MoveL Offs(pOrigin,43.1,66.3,0.0),vDraw,z1,tPen\WObj:=wPaper;
    MoveL Offs(pOrigin,43.4,66.5,0.0),vDraw,z1,tPen\WObj:=wPaper;
    MoveL Offs(pOrigin,43.4,67.1,0.0),vDraw,z1,tPen\WObj:=wPaper;
    MoveL Offs(pOrigin,43.7,67.3,0.0),vDraw,z1,tPen\WObj:=wPaper;
    MoveL Offs(pOrigin,43.7,67.9,0.0),vDraw,z1,tPen\WObj:=wPaper;
    MoveL Offs(pOrigin,43.9,68.1,0.0),vDraw,z1,tPen\WObj:=wPaper;
    MoveL Offs(pOrigin,44.2,68.1,0.0),vDraw,z1,tPen\WObj:=wPaper;
    MoveL Offs(pOrigin,44.5,68.4,0.0),vDraw,z1,tPen\WObj:=wPaper;
    MoveL Offs(pOrigin,56.7,68.4,0.0),vDraw,z1,tPen\WObj:=wPaper;
    MoveL Offs(pOrigin,57.0,68.7,0.0),vDraw,z1,tPen\WObj:=wPaper;
    MoveL Offs(pOrigin,57.0,90.3,0.0),vDraw,fine,tPen\WObj:=wPaper;
    MoveL Offs(pOrigin,57.0,90.3,15.0),vApproach,z5,tPen\WObj:=wPaper;
    MoveL Offs(pOrigin,107.1,90.3,15.0),vTravel,z5,tPen\WObj:=wPaper;
    MoveL Offs(pOrigin,107.1,90.3,0.0),vApproach,fine,tPen\WObj:=wPaper;
    MoveL Offs(pOrigin,107.1,51.1,0.0),vDraw,z1,tPen\WObj:=wPaper;
    MoveL Offs(pOrigin,107.4,50.8,0.0),vDraw,z1,tPen\WObj:=wPaper;
    MoveL Offs(pOrigin,131.9,50.8,0.0),vDraw,z1,tPen\WObj:=wPaper;
    MoveL Offs(pOrigin,131.9,90.3,0.0),vDraw,z1,tPen\WObj:=wPaper;
    MoveL Offs(pOrigin,131.7,90.5,0.0),vDraw,z1,tPen\WObj:=wPaper;
    MoveL Offs(pOrigin,125.5,90.5,0.0),vDraw,z1,tPen\WObj:=wPaper;
    MoveL Offs(pOrigin,125.3,90.3,0.0),vDraw,z1,tPen\WObj:=wPaper;
    MoveL Offs(pOrigin,125.0,90.3,0.0),vDraw,z1,tPen\WObj:=wPaper;
    MoveL Offs(pOrigin,124.7,90.5,0.0),vDraw,z1,tPen\WObj:=wPaper;
    MoveL Offs(pOrigin,112.7,90.5,0.0),vDraw,z1,tPen\WObj:=wPaper;
    MoveL Offs(pOrigin,112.5,90.3,0.0),vDraw,z1,tPen\WObj:=wPaper;
    MoveL Offs(pOrigin,111.9,90.3,0.0),vDraw,z1,tPen\WObj:=wPaper;
    MoveL Offs(pOrigin,111.7,90.5,0.0),vDraw,z1,tPen\WObj:=wPaper;
    MoveL Offs(pOrigin,107.4,90.5,0.0),vDraw,z1,tPen\WObj:=wPaper;
    MoveL Offs(pOrigin,107.1,90.3,0.0),vDraw,fine,tPen\WObj:=wPaper;
    MoveL Offs(pOrigin,107.1,90.3,15.0),vApproach,z5,tPen\WObj:=wPaper;
    MoveL Offs(pOrigin,107.7,92.9,15.0),vTravel,z5,tPen\WObj:=wPaper;
    MoveL Offs(pOrigin,107.7,92.9,0.0),vApproach,fine,tPen\WObj:=wPaper;
    MoveL Offs(pOrigin,114.3,92.9,0.0),vDraw,z1,tPen\WObj:=wPaper;
    MoveL Offs(pOrigin,114.6,93.2,0.0),vDraw,z1,tPen\WObj:=wPaper;
    MoveL Offs(pOrigin,115.4,93.2,0.0),vDraw,z1,tPen\WObj:=wPaper;
    MoveL Offs(pOrigin,115.7,92.9,0.0),vDraw,z1,tPen\WObj:=wPaper;
    MoveL Offs(pOrigin,116.7,92.9,0.0),vDraw,z1,tPen\WObj:=wPaper;
    MoveL Offs(pOrigin,117.0,93.2,0.0),vDraw,z1,tPen\WObj:=wPaper;
    MoveL Offs(pOrigin,117.3,92.9,0.0),vDraw,z1,tPen\WObj:=wPaper;
    MoveL Offs(pOrigin,129.8,92.9,0.0),vDraw,z1,tPen\WObj:=wPaper;
    MoveL Offs(pOrigin,130.1,93.2,0.0),vDraw,z1,tPen\WObj:=wPaper;
    MoveL Offs(pOrigin,130.3,92.9,0.0),vDraw,z1,tPen\WObj:=wPaper;
    MoveL Offs(pOrigin,131.7,92.9,0.0),vDraw,z1,tPen\WObj:=wPaper;
    MoveL Offs(pOrigin,131.9,93.2,0.0),vDraw,z1,tPen\WObj:=wPaper;
    MoveL Offs(pOrigin,131.9,132.9,0.0),vDraw,z1,tPen\WObj:=wPaper;
    MoveL Offs(pOrigin,131.7,133.2,0.0),vDraw,z1,tPen\WObj:=wPaper;
    MoveL Offs(pOrigin,107.4,133.2,0.0),vDraw,z1,tPen\WObj:=wPaper;
    MoveL Offs(pOrigin,107.1,132.9,0.0),vDraw,z1,tPen\WObj:=wPaper;
    MoveL Offs(pOrigin,107.1,93.2,0.0),vDraw,z1,tPen\WObj:=wPaper;
    MoveL Offs(pOrigin,107.4,93.2,0.0),vDraw,z1,tPen\WObj:=wPaper;
    MoveL Offs(pOrigin,107.7,92.9,0.0),vDraw,fine,tPen\WObj:=wPaper;
    MoveL Offs(pOrigin,107.7,92.9,15.0),vApproach,z5,tPen\WObj:=wPaper;
  ENDPROC

  PROC Part5()
    MoveL Offs(pOrigin,134.6,93.2,15.0),vTravel,z5,tPen\WObj:=wPaper;
    MoveL Offs(pOrigin,134.6,93.2,0.0),vApproach,fine,tPen\WObj:=wPaper;
    MoveL Offs(pOrigin,134.9,93.2,0.0),vDraw,z1,tPen\WObj:=wPaper;
    MoveL Offs(pOrigin,135.1,92.9,0.0),vDraw,z1,tPen\WObj:=wPaper;
    MoveL Offs(pOrigin,142.6,92.9,0.0),vDraw,z1,tPen\WObj:=wPaper;
    MoveL Offs(pOrigin,142.9,93.2,0.0),vDraw,z1,tPen\WObj:=wPaper;
    MoveL Offs(pOrigin,143.1,93.2,0.0),vDraw,z1,tPen\WObj:=wPaper;
    MoveL Offs(pOrigin,143.4,92.9,0.0),vDraw,z1,tPen\WObj:=wPaper;
    MoveL Offs(pOrigin,159.4,92.9,0.0),vDraw,z1,tPen\WObj:=wPaper;
    MoveL Offs(pOrigin,159.7,93.2,0.0),vDraw,z1,tPen\WObj:=wPaper;
    MoveL Offs(pOrigin,159.7,93.5,0.0),vDraw,z1,tPen\WObj:=wPaper;
    MoveL Offs(pOrigin,155.7,97.5,0.0),vDraw,z1,tPen\WObj:=wPaper;
    MoveL Offs(pOrigin,155.4,97.5,0.0),vDraw,z1,tPen\WObj:=wPaper;
    MoveL Offs(pOrigin,154.6,98.3,0.0),vDraw,z1,tPen\WObj:=wPaper;
    MoveL Offs(pOrigin,154.3,98.3,0.0),vDraw,z1,tPen\WObj:=wPaper;
    MoveL Offs(pOrigin,153.5,99.1,0.0),vDraw,z1,tPen\WObj:=wPaper;
    MoveL Offs(pOrigin,153.3,99.1,0.0),vDraw,z1,tPen\WObj:=wPaper;
    MoveL Offs(pOrigin,151.9,100.1,0.0),vDraw,z1,tPen\WObj:=wPaper;
    MoveL Offs(pOrigin,151.1,100.4,0.0),vDraw,z1,tPen\WObj:=wPaper;
    MoveL Offs(pOrigin,150.3,101.2,0.0),vDraw,z1,tPen\WObj:=wPaper;
    MoveL Offs(pOrigin,150.3,101.5,0.0),vDraw,z1,tPen\WObj:=wPaper;
    MoveL Offs(pOrigin,151.1,102.3,0.0),vDraw,z1,tPen\WObj:=wPaper;
    MoveL Offs(pOrigin,151.4,102.3,0.0),vDraw,z1,tPen\WObj:=wPaper;
    MoveL Offs(pOrigin,154.1,104.9,0.0),vDraw,z1,tPen\WObj:=wPaper;
    MoveL Offs(pOrigin,154.1,105.2,0.0),vDraw,z1,tPen\WObj:=wPaper;
    MoveL Offs(pOrigin,155.4,106.8,0.0),vDraw,z1,tPen\WObj:=wPaper;
    MoveL Offs(pOrigin,155.4,107.1,0.0),vDraw,z1,tPen\WObj:=wPaper;
    MoveL Offs(pOrigin,156.5,108.9,0.0),vDraw,z1,tPen\WObj:=wPaper;
    MoveL Offs(pOrigin,156.5,109.5,0.0),vDraw,z1,tPen\WObj:=wPaper;
    MoveL Offs(pOrigin,156.7,109.7,0.0),vDraw,z1,tPen\WObj:=wPaper;
    MoveL Offs(pOrigin,156.7,110.3,0.0),vDraw,z1,tPen\WObj:=wPaper;
    MoveL Offs(pOrigin,157.0,110.5,0.0),vDraw,z1,tPen\WObj:=wPaper;
    MoveL Offs(pOrigin,157.0,111.1,0.0),vDraw,z1,tPen\WObj:=wPaper;
    MoveL Offs(pOrigin,157.3,111.3,0.0),vDraw,z1,tPen\WObj:=wPaper;
    MoveL Offs(pOrigin,157.3,112.1,0.0),vDraw,z1,tPen\WObj:=wPaper;
    MoveL Offs(pOrigin,157.5,112.4,0.0),vDraw,z1,tPen\WObj:=wPaper;
    MoveL Offs(pOrigin,157.5,118.8,0.0),vDraw,z1,tPen\WObj:=wPaper;
    MoveL Offs(pOrigin,157.3,119.1,0.0),vDraw,z1,tPen\WObj:=wPaper;
    MoveL Offs(pOrigin,157.3,119.9,0.0),vDraw,z1,tPen\WObj:=wPaper;
    MoveL Offs(pOrigin,157.0,120.1,0.0),vDraw,z1,tPen\WObj:=wPaper;
    MoveL Offs(pOrigin,157.0,120.7,0.0),vDraw,z1,tPen\WObj:=wPaper;
    MoveL Offs(pOrigin,156.7,120.9,0.0),vDraw,z1,tPen\WObj:=wPaper;
    MoveL Offs(pOrigin,156.5,122.3,0.0),vDraw,z1,tPen\WObj:=wPaper;
    MoveL Offs(pOrigin,156.2,122.5,0.0),vDraw,z1,tPen\WObj:=wPaper;
    MoveL Offs(pOrigin,155.4,124.4,0.0),vDraw,z1,tPen\WObj:=wPaper;
    MoveL Offs(pOrigin,154.9,124.9,0.0),vDraw,z1,tPen\WObj:=wPaper;
    MoveL Offs(pOrigin,154.9,125.2,0.0),vDraw,z1,tPen\WObj:=wPaper;
    MoveL Offs(pOrigin,154.3,125.7,0.0),vDraw,z1,tPen\WObj:=wPaper;
    MoveL Offs(pOrigin,154.3,126.0,0.0),vDraw,z1,tPen\WObj:=wPaper;
    MoveL Offs(pOrigin,153.3,127.1,0.0),vDraw,z1,tPen\WObj:=wPaper;
    MoveL Offs(pOrigin,153.3,127.3,0.0),vDraw,z1,tPen\WObj:=wPaper;
    MoveL Offs(pOrigin,151.9,128.7,0.0),vDraw,z1,tPen\WObj:=wPaper;
    MoveL Offs(pOrigin,151.7,128.7,0.0),vDraw,z1,tPen\WObj:=wPaper;
    MoveL Offs(pOrigin,149.5,130.5,0.0),vDraw,z1,tPen\WObj:=wPaper;
    MoveL Offs(pOrigin,149.3,130.5,0.0),vDraw,z1,tPen\WObj:=wPaper;
    MoveL Offs(pOrigin,146.3,132.1,0.0),vDraw,z1,tPen\WObj:=wPaper;
    MoveL Offs(pOrigin,145.8,132.1,0.0),vDraw,z1,tPen\WObj:=wPaper;
    MoveL Offs(pOrigin,145.5,132.4,0.0),vDraw,z1,tPen\WObj:=wPaper;
    MoveL Offs(pOrigin,145.0,132.4,0.0),vDraw,z1,tPen\WObj:=wPaper;
    MoveL Offs(pOrigin,144.7,132.7,0.0),vDraw,z1,tPen\WObj:=wPaper;
    MoveL Offs(pOrigin,143.9,132.7,0.0),vDraw,z1,tPen\WObj:=wPaper;
    MoveL Offs(pOrigin,143.7,132.9,0.0),vDraw,z1,tPen\WObj:=wPaper;
    MoveL Offs(pOrigin,142.1,132.9,0.0),vDraw,z1,tPen\WObj:=wPaper;
    MoveL Offs(pOrigin,141.8,133.2,0.0),vDraw,z1,tPen\WObj:=wPaper;
    MoveL Offs(pOrigin,135.1,133.2,0.0),vDraw,z1,tPen\WObj:=wPaper;
    MoveL Offs(pOrigin,134.9,132.9,0.0),vDraw,z1,tPen\WObj:=wPaper;
    MoveL Offs(pOrigin,134.6,132.9,0.0),vDraw,z1,tPen\WObj:=wPaper;
    MoveL Offs(pOrigin,134.6,93.2,0.0),vDraw,fine,tPen\WObj:=wPaper;
    MoveL Offs(pOrigin,134.6,93.2,15.0),vApproach,z5,tPen\WObj:=wPaper;
    MoveL Offs(pOrigin,135.1,90.5,15.0),vTravel,z5,tPen\WObj:=wPaper;
    MoveL Offs(pOrigin,135.1,90.5,0.0),vApproach,fine,tPen\WObj:=wPaper;
    MoveL Offs(pOrigin,134.6,90.0,0.0),vDraw,z1,tPen\WObj:=wPaper;
    MoveL Offs(pOrigin,134.6,51.1,0.0),vDraw,z1,tPen\WObj:=wPaper;
    MoveL Offs(pOrigin,134.9,50.8,0.0),vDraw,z1,tPen\WObj:=wPaper;
    MoveL Offs(pOrigin,141.5,50.8,0.0),vDraw,z1,tPen\WObj:=wPaper;
    MoveL Offs(pOrigin,141.8,51.1,0.0),vDraw,z1,tPen\WObj:=wPaper;
    MoveL Offs(pOrigin,143.1,51.1,0.0),vDraw,z1,tPen\WObj:=wPaper;
    MoveL Offs(pOrigin,143.4,51.3,0.0),vDraw,z1,tPen\WObj:=wPaper;
    MoveL Offs(pOrigin,144.5,51.3,0.0),vDraw,z1,tPen\WObj:=wPaper;
    MoveL Offs(pOrigin,144.7,51.6,0.0),vDraw,z1,tPen\WObj:=wPaper;
    MoveL Offs(pOrigin,145.5,51.6,0.0),vDraw,z1,tPen\WObj:=wPaper;
    MoveL Offs(pOrigin,145.8,51.9,0.0),vDraw,z1,tPen\WObj:=wPaper;
    MoveL Offs(pOrigin,146.6,51.9,0.0),vDraw,z1,tPen\WObj:=wPaper;
    MoveL Offs(pOrigin,146.9,52.1,0.0),vDraw,z1,tPen\WObj:=wPaper;
    MoveL Offs(pOrigin,148.2,52.4,0.0),vDraw,z1,tPen\WObj:=wPaper;
    MoveL Offs(pOrigin,148.5,52.7,0.0),vDraw,z1,tPen\WObj:=wPaper;
    MoveL Offs(pOrigin,148.7,52.7,0.0),vDraw,z1,tPen\WObj:=wPaper;
    MoveL Offs(pOrigin,149.0,52.9,0.0),vDraw,z1,tPen\WObj:=wPaper;
    MoveL Offs(pOrigin,149.3,52.9,0.0),vDraw,z1,tPen\WObj:=wPaper;
    MoveL Offs(pOrigin,149.5,53.2,0.0),vDraw,z1,tPen\WObj:=wPaper;
    MoveL Offs(pOrigin,149.8,53.2,0.0),vDraw,z1,tPen\WObj:=wPaper;
    MoveL Offs(pOrigin,150.1,53.5,0.0),vDraw,z1,tPen\WObj:=wPaper;
    MoveL Offs(pOrigin,150.3,53.5,0.0),vDraw,z1,tPen\WObj:=wPaper;
    MoveL Offs(pOrigin,150.6,53.7,0.0),vDraw,z1,tPen\WObj:=wPaper;
    MoveL Offs(pOrigin,152.5,54.5,0.0),vDraw,z1,tPen\WObj:=wPaper;
    MoveL Offs(pOrigin,153.0,55.1,0.0),vDraw,z1,tPen\WObj:=wPaper;
    MoveL Offs(pOrigin,153.3,55.1,0.0),vDraw,z1,tPen\WObj:=wPaper;
    MoveL Offs(pOrigin,153.8,55.6,0.0),vDraw,z1,tPen\WObj:=wPaper;
    MoveL Offs(pOrigin,154.1,55.6,0.0),vDraw,z1,tPen\WObj:=wPaper;
    MoveL Offs(pOrigin,154.9,56.4,0.0),vDraw,z1,tPen\WObj:=wPaper;
    MoveL Offs(pOrigin,155.1,56.4,0.0),vDraw,z1,tPen\WObj:=wPaper;
    MoveL Offs(pOrigin,157.0,58.3,0.0),vDraw,z1,tPen\WObj:=wPaper;
    MoveL Offs(pOrigin,157.3,58.3,0.0),vDraw,z1,tPen\WObj:=wPaper;
    MoveL Offs(pOrigin,157.5,58.5,0.0),vDraw,z1,tPen\WObj:=wPaper;
    MoveL Offs(pOrigin,157.5,58.8,0.0),vDraw,z1,tPen\WObj:=wPaper;
    MoveL Offs(pOrigin,159.4,60.7,0.0),vDraw,z1,tPen\WObj:=wPaper;
    MoveL Offs(pOrigin,159.4,60.9,0.0),vDraw,z1,tPen\WObj:=wPaper;
    MoveL Offs(pOrigin,160.7,62.5,0.0),vDraw,z1,tPen\WObj:=wPaper;
    MoveL Offs(pOrigin,160.7,62.8,0.0),vDraw,z1,tPen\WObj:=wPaper;
    MoveL Offs(pOrigin,161.5,63.9,0.0),vDraw,z1,tPen\WObj:=wPaper;
    MoveL Offs(pOrigin,161.5,64.1,0.0),vDraw,z1,tPen\WObj:=wPaper;
    MoveL Offs(pOrigin,162.9,66.5,0.0),vDraw,z1,tPen\WObj:=wPaper;
    MoveL Offs(pOrigin,162.9,67.1,0.0),vDraw,z1,tPen\WObj:=wPaper;
    MoveL Offs(pOrigin,163.4,67.9,0.0),vDraw,z1,tPen\WObj:=wPaper;
    MoveL Offs(pOrigin,163.4,68.4,0.0),vDraw,z1,tPen\WObj:=wPaper;
    MoveL Offs(pOrigin,163.7,68.7,0.0),vDraw,z1,tPen\WObj:=wPaper;
    MoveL Offs(pOrigin,163.7,69.2,0.0),vDraw,z1,tPen\WObj:=wPaper;
    MoveL Offs(pOrigin,163.9,69.5,0.0),vDraw,z1,tPen\WObj:=wPaper;
    MoveL Offs(pOrigin,163.9,70.3,0.0),vDraw,z1,tPen\WObj:=wPaper;
    MoveL Offs(pOrigin,164.2,70.5,0.0),vDraw,z1,tPen\WObj:=wPaper;
  ENDPROC

  PROC Part6()
    MoveL Offs(pOrigin,164.2,71.3,0.0),vDraw,z1,tPen\WObj:=wPaper;
    MoveL Offs(pOrigin,164.5,71.6,0.0),vDraw,z1,tPen\WObj:=wPaper;
    MoveL Offs(pOrigin,164.5,73.2,0.0),vDraw,z1,tPen\WObj:=wPaper;
    MoveL Offs(pOrigin,164.7,73.5,0.0),vDraw,z1,tPen\WObj:=wPaper;
    MoveL Offs(pOrigin,164.7,75.1,0.0),vDraw,z1,tPen\WObj:=wPaper;
    MoveL Offs(pOrigin,165.0,75.3,0.0),vDraw,z1,tPen\WObj:=wPaper;
    MoveL Offs(pOrigin,165.0,78.8,0.0),vDraw,z1,tPen\WObj:=wPaper;
    MoveL Offs(pOrigin,164.7,79.1,0.0),vDraw,z1,tPen\WObj:=wPaper;
    MoveL Offs(pOrigin,164.7,82.3,0.0),vDraw,z1,tPen\WObj:=wPaper;
    MoveL Offs(pOrigin,164.5,82.5,0.0),vDraw,z1,tPen\WObj:=wPaper;
    MoveL Offs(pOrigin,164.5,83.6,0.0),vDraw,z1,tPen\WObj:=wPaper;
    MoveL Offs(pOrigin,164.2,83.9,0.0),vDraw,z1,tPen\WObj:=wPaper;
    MoveL Offs(pOrigin,164.2,84.7,0.0),vDraw,z1,tPen\WObj:=wPaper;
    MoveL Offs(pOrigin,163.9,84.9,0.0),vDraw,z1,tPen\WObj:=wPaper;
    MoveL Offs(pOrigin,163.7,86.3,0.0),vDraw,z1,tPen\WObj:=wPaper;
    MoveL Offs(pOrigin,163.1,87.1,0.0),vDraw,z1,tPen\WObj:=wPaper;
    MoveL Offs(pOrigin,163.1,87.6,0.0),vDraw,z1,tPen\WObj:=wPaper;
    MoveL Offs(pOrigin,162.9,87.9,0.0),vDraw,z1,tPen\WObj:=wPaper;
    MoveL Offs(pOrigin,162.1,89.7,0.0),vDraw,z1,tPen\WObj:=wPaper;
    MoveL Offs(pOrigin,161.3,90.5,0.0),vDraw,z1,tPen\WObj:=wPaper;
    MoveL Offs(pOrigin,135.1,90.5,0.0),vDraw,fine,tPen\WObj:=wPaper;
    MoveL Offs(pOrigin,135.1,90.5,15.0),vApproach,z5,tPen\WObj:=wPaper;
    MoveL Offs(pOrigin,174.3,90.0,15.0),vTravel,z5,tPen\WObj:=wPaper;
    MoveL Offs(pOrigin,174.3,90.0,0.0),vApproach,fine,tPen\WObj:=wPaper;
    MoveL Offs(pOrigin,174.3,51.1,0.0),vDraw,z1,tPen\WObj:=wPaper;
    MoveL Offs(pOrigin,174.6,50.8,0.0),vDraw,z1,tPen\WObj:=wPaper;
    MoveL Offs(pOrigin,198.9,50.8,0.0),vDraw,z1,tPen\WObj:=wPaper;
    MoveL Offs(pOrigin,199.1,51.1,0.0),vDraw,z1,tPen\WObj:=wPaper;
    MoveL Offs(pOrigin,199.1,53.2,0.0),vDraw,z1,tPen\WObj:=wPaper;
    MoveL Offs(pOrigin,199.4,53.5,0.0),vDraw,z1,tPen\WObj:=wPaper;
    MoveL Offs(pOrigin,199.4,58.0,0.0),vDraw,z1,tPen\WObj:=wPaper;
    MoveL Offs(pOrigin,199.1,58.3,0.0),vDraw,z1,tPen\WObj:=wPaper;
    MoveL Offs(pOrigin,199.1,59.1,0.0),vDraw,z1,tPen\WObj:=wPaper;
    MoveL Offs(pOrigin,199.4,59.3,0.0),vDraw,z1,tPen\WObj:=wPaper;
    MoveL Offs(pOrigin,199.4,59.9,0.0),vDraw,z1,tPen\WObj:=wPaper;
    MoveL Offs(pOrigin,199.1,60.1,0.0),vDraw,z1,tPen\WObj:=wPaper;
    MoveL Offs(pOrigin,199.4,60.4,0.0),vDraw,z1,tPen\WObj:=wPaper;
    MoveL Offs(pOrigin,199.4,64.7,0.0),vDraw,z1,tPen\WObj:=wPaper;
    MoveL Offs(pOrigin,199.1,64.9,0.0),vDraw,z1,tPen\WObj:=wPaper;
    MoveL Offs(pOrigin,199.1,67.6,0.0),vDraw,z1,tPen\WObj:=wPaper;
    MoveL Offs(pOrigin,199.4,67.9,0.0),vDraw,z1,tPen\WObj:=wPaper;
    MoveL Offs(pOrigin,199.4,73.7,0.0),vDraw,z1,tPen\WObj:=wPaper;
    MoveL Offs(pOrigin,199.1,74.0,0.0),vDraw,z1,tPen\WObj:=wPaper;
    MoveL Offs(pOrigin,199.1,74.3,0.0),vDraw,z1,tPen\WObj:=wPaper;
    MoveL Offs(pOrigin,199.4,74.5,0.0),vDraw,z1,tPen\WObj:=wPaper;
    MoveL Offs(pOrigin,199.4,78.5,0.0),vDraw,z1,tPen\WObj:=wPaper;
    MoveL Offs(pOrigin,199.1,78.8,0.0),vDraw,z1,tPen\WObj:=wPaper;
    MoveL Offs(pOrigin,199.1,79.1,0.0),vDraw,z1,tPen\WObj:=wPaper;
    MoveL Offs(pOrigin,199.4,79.3,0.0),vDraw,z1,tPen\WObj:=wPaper;
    MoveL Offs(pOrigin,199.4,79.9,0.0),vDraw,z1,tPen\WObj:=wPaper;
    MoveL Offs(pOrigin,199.1,80.1,0.0),vDraw,z1,tPen\WObj:=wPaper;
    MoveL Offs(pOrigin,199.1,81.2,0.0),vDraw,z1,tPen\WObj:=wPaper;
    MoveL Offs(pOrigin,199.4,81.5,0.0),vDraw,z1,tPen\WObj:=wPaper;
    MoveL Offs(pOrigin,199.4,85.5,0.0),vDraw,z1,tPen\WObj:=wPaper;
    MoveL Offs(pOrigin,199.1,85.7,0.0),vDraw,z1,tPen\WObj:=wPaper;
    MoveL Offs(pOrigin,199.1,88.4,0.0),vDraw,z1,tPen\WObj:=wPaper;
    MoveL Offs(pOrigin,199.4,88.7,0.0),vDraw,z1,tPen\WObj:=wPaper;
    MoveL Offs(pOrigin,199.4,90.0,0.0),vDraw,z1,tPen\WObj:=wPaper;
    MoveL Offs(pOrigin,198.9,90.5,0.0),vDraw,z1,tPen\WObj:=wPaper;
    MoveL Offs(pOrigin,190.1,90.5,0.0),vDraw,z1,tPen\WObj:=wPaper;
    MoveL Offs(pOrigin,189.8,90.3,0.0),vDraw,z1,tPen\WObj:=wPaper;
    MoveL Offs(pOrigin,189.3,90.3,0.0),vDraw,z1,tPen\WObj:=wPaper;
    MoveL Offs(pOrigin,189.0,90.5,0.0),vDraw,z1,tPen\WObj:=wPaper;
    MoveL Offs(pOrigin,177.0,90.5,0.0),vDraw,z1,tPen\WObj:=wPaper;
    MoveL Offs(pOrigin,176.7,90.3,0.0),vDraw,z1,tPen\WObj:=wPaper;
    MoveL Offs(pOrigin,176.2,90.3,0.0),vDraw,z1,tPen\WObj:=wPaper;
    MoveL Offs(pOrigin,175.9,90.5,0.0),vDraw,z1,tPen\WObj:=wPaper;
    MoveL Offs(pOrigin,174.9,90.5,0.0),vDraw,z1,tPen\WObj:=wPaper;
    MoveL Offs(pOrigin,174.3,90.0,0.0),vDraw,fine,tPen\WObj:=wPaper;
    MoveL Offs(pOrigin,174.3,90.0,15.0),vApproach,z5,tPen\WObj:=wPaper;
    MoveL Offs(pOrigin,174.9,92.9,15.0),vTravel,z5,tPen\WObj:=wPaper;
    MoveL Offs(pOrigin,174.9,92.9,0.0),vApproach,fine,tPen\WObj:=wPaper;
    MoveL Offs(pOrigin,178.9,92.9,0.0),vDraw,z1,tPen\WObj:=wPaper;
    MoveL Offs(pOrigin,179.1,93.2,0.0),vDraw,z1,tPen\WObj:=wPaper;
    MoveL Offs(pOrigin,179.7,93.2,0.0),vDraw,z1,tPen\WObj:=wPaper;
    MoveL Offs(pOrigin,179.9,92.9,0.0),vDraw,z1,tPen\WObj:=wPaper;
    MoveL Offs(pOrigin,191.7,92.9,0.0),vDraw,z1,tPen\WObj:=wPaper;
    MoveL Offs(pOrigin,191.9,93.2,0.0),vDraw,z1,tPen\WObj:=wPaper;
    MoveL Offs(pOrigin,192.7,93.2,0.0),vDraw,z1,tPen\WObj:=wPaper;
    MoveL Offs(pOrigin,193.0,92.9,0.0),vDraw,z1,tPen\WObj:=wPaper;
    MoveL Offs(pOrigin,198.6,92.9,0.0),vDraw,z1,tPen\WObj:=wPaper;
    MoveL Offs(pOrigin,198.9,93.2,0.0),vDraw,z1,tPen\WObj:=wPaper;
    MoveL Offs(pOrigin,199.1,93.2,0.0),vDraw,z1,tPen\WObj:=wPaper;
    MoveL Offs(pOrigin,199.1,95.6,0.0),vDraw,z1,tPen\WObj:=wPaper;
    MoveL Offs(pOrigin,199.4,95.9,0.0),vDraw,z1,tPen\WObj:=wPaper;
    MoveL Offs(pOrigin,199.4,99.6,0.0),vDraw,z1,tPen\WObj:=wPaper;
    MoveL Offs(pOrigin,199.1,99.9,0.0),vDraw,z1,tPen\WObj:=wPaper;
    MoveL Offs(pOrigin,199.1,102.8,0.0),vDraw,z1,tPen\WObj:=wPaper;
    MoveL Offs(pOrigin,199.4,103.1,0.0),vDraw,z1,tPen\WObj:=wPaper;
    MoveL Offs(pOrigin,199.4,106.8,0.0),vDraw,z1,tPen\WObj:=wPaper;
    MoveL Offs(pOrigin,199.1,107.1,0.0),vDraw,z1,tPen\WObj:=wPaper;
    MoveL Offs(pOrigin,199.1,109.5,0.0),vDraw,z1,tPen\WObj:=wPaper;
    MoveL Offs(pOrigin,199.4,109.7,0.0),vDraw,z1,tPen\WObj:=wPaper;
    MoveL Offs(pOrigin,199.4,114.0,0.0),vDraw,z1,tPen\WObj:=wPaper;
    MoveL Offs(pOrigin,199.1,114.3,0.0),vDraw,z1,tPen\WObj:=wPaper;
    MoveL Offs(pOrigin,199.1,116.4,0.0),vDraw,z1,tPen\WObj:=wPaper;
    MoveL Offs(pOrigin,199.4,116.7,0.0),vDraw,z1,tPen\WObj:=wPaper;
    MoveL Offs(pOrigin,199.4,120.9,0.0),vDraw,z1,tPen\WObj:=wPaper;
    MoveL Offs(pOrigin,199.1,121.2,0.0),vDraw,z1,tPen\WObj:=wPaper;
    MoveL Offs(pOrigin,199.1,123.9,0.0),vDraw,z1,tPen\WObj:=wPaper;
    MoveL Offs(pOrigin,199.4,124.1,0.0),vDraw,z1,tPen\WObj:=wPaper;
    MoveL Offs(pOrigin,199.4,128.1,0.0),vDraw,z1,tPen\WObj:=wPaper;
    MoveL Offs(pOrigin,199.1,128.4,0.0),vDraw,z1,tPen\WObj:=wPaper;
    MoveL Offs(pOrigin,199.1,130.5,0.0),vDraw,z1,tPen\WObj:=wPaper;
    MoveL Offs(pOrigin,199.4,130.8,0.0),vDraw,z1,tPen\WObj:=wPaper;
    MoveL Offs(pOrigin,199.4,132.7,0.0),vDraw,z1,tPen\WObj:=wPaper;
    MoveL Offs(pOrigin,198.9,133.2,0.0),vDraw,z1,tPen\WObj:=wPaper;
    MoveL Offs(pOrigin,174.9,133.2,0.0),vDraw,z1,tPen\WObj:=wPaper;
    MoveL Offs(pOrigin,174.3,132.7,0.0),vDraw,z1,tPen\WObj:=wPaper;
    MoveL Offs(pOrigin,174.3,93.2,0.0),vDraw,z1,tPen\WObj:=wPaper;
    MoveL Offs(pOrigin,174.6,93.2,0.0),vDraw,z1,tPen\WObj:=wPaper;
    MoveL Offs(pOrigin,174.9,92.9,0.0),vDraw,fine,tPen\WObj:=wPaper;
    MoveL Offs(pOrigin,174.9,92.9,15.0),vApproach,z5,tPen\WObj:=wPaper;
    MoveL Offs(pOrigin,202.1,93.2,15.0),vTravel,z5,tPen\WObj:=wPaper;
    MoveL Offs(pOrigin,202.1,93.2,0.0),vApproach,fine,tPen\WObj:=wPaper;
    MoveL Offs(pOrigin,202.3,92.9,0.0),vDraw,z1,tPen\WObj:=wPaper;
    MoveL Offs(pOrigin,207.1,92.9,0.0),vDraw,z1,tPen\WObj:=wPaper;
    MoveL Offs(pOrigin,207.4,93.2,0.0),vDraw,z1,tPen\WObj:=wPaper;
    MoveL Offs(pOrigin,207.7,92.9,0.0),vDraw,z1,tPen\WObj:=wPaper;
    MoveL Offs(pOrigin,219.9,92.9,0.0),vDraw,z1,tPen\WObj:=wPaper;
  ENDPROC

  PROC Part7()
    MoveL Offs(pOrigin,220.2,93.2,0.0),vDraw,z1,tPen\WObj:=wPaper;
    MoveL Offs(pOrigin,220.5,93.2,0.0),vDraw,z1,tPen\WObj:=wPaper;
    MoveL Offs(pOrigin,220.7,92.9,0.0),vDraw,z1,tPen\WObj:=wPaper;
    MoveL Offs(pOrigin,226.6,92.9,0.0),vDraw,z1,tPen\WObj:=wPaper;
    MoveL Offs(pOrigin,226.9,93.2,0.0),vDraw,z1,tPen\WObj:=wPaper;
    MoveL Offs(pOrigin,227.1,93.2,0.0),vDraw,z1,tPen\WObj:=wPaper;
    MoveL Offs(pOrigin,226.3,94.0,0.0),vDraw,z1,tPen\WObj:=wPaper;
    MoveL Offs(pOrigin,226.3,94.3,0.0),vDraw,z1,tPen\WObj:=wPaper;
    MoveL Offs(pOrigin,222.3,98.0,0.0),vDraw,z1,tPen\WObj:=wPaper;
    MoveL Offs(pOrigin,222.1,98.0,0.0),vDraw,z1,tPen\WObj:=wPaper;
    MoveL Offs(pOrigin,221.3,98.8,0.0),vDraw,z1,tPen\WObj:=wPaper;
    MoveL Offs(pOrigin,221.0,98.8,0.0),vDraw,z1,tPen\WObj:=wPaper;
    MoveL Offs(pOrigin,218.9,100.4,0.0),vDraw,z1,tPen\WObj:=wPaper;
    MoveL Offs(pOrigin,218.1,100.7,0.0),vDraw,z1,tPen\WObj:=wPaper;
    MoveL Offs(pOrigin,217.5,101.2,0.0),vDraw,z1,tPen\WObj:=wPaper;
    MoveL Offs(pOrigin,219.7,103.3,0.0),vDraw,z1,tPen\WObj:=wPaper;
    MoveL Offs(pOrigin,219.9,103.3,0.0),vDraw,z1,tPen\WObj:=wPaper;
    MoveL Offs(pOrigin,220.7,104.1,0.0),vDraw,z1,tPen\WObj:=wPaper;
    MoveL Offs(pOrigin,220.7,104.4,0.0),vDraw,z1,tPen\WObj:=wPaper;
    MoveL Offs(pOrigin,221.8,105.5,0.0),vDraw,z1,tPen\WObj:=wPaper;
    MoveL Offs(pOrigin,221.8,105.7,0.0),vDraw,z1,tPen\WObj:=wPaper;
    MoveL Offs(pOrigin,222.9,107.1,0.0),vDraw,z1,tPen\WObj:=wPaper;
    MoveL Offs(pOrigin,222.9,107.3,0.0),vDraw,z1,tPen\WObj:=wPaper;
    MoveL Offs(pOrigin,223.7,108.7,0.0),vDraw,z1,tPen\WObj:=wPaper;
    MoveL Offs(pOrigin,223.7,109.2,0.0),vDraw,z1,tPen\WObj:=wPaper;
    MoveL Offs(pOrigin,224.2,110.0,0.0),vDraw,z1,tPen\WObj:=wPaper;
    MoveL Offs(pOrigin,224.2,110.8,0.0),vDraw,z1,tPen\WObj:=wPaper;
    MoveL Offs(pOrigin,224.5,111.1,0.0),vDraw,z1,tPen\WObj:=wPaper;
    MoveL Offs(pOrigin,224.5,111.9,0.0),vDraw,z1,tPen\WObj:=wPaper;
    MoveL Offs(pOrigin,224.7,112.1,0.0),vDraw,z1,tPen\WObj:=wPaper;
    MoveL Offs(pOrigin,224.7,113.5,0.0),vDraw,z1,tPen\WObj:=wPaper;
    MoveL Offs(pOrigin,225.0,113.7,0.0),vDraw,z1,tPen\WObj:=wPaper;
    MoveL Offs(pOrigin,225.0,117.2,0.0),vDraw,z1,tPen\WObj:=wPaper;
    MoveL Offs(pOrigin,224.7,117.5,0.0),vDraw,z1,tPen\WObj:=wPaper;
    MoveL Offs(pOrigin,224.7,119.1,0.0),vDraw,z1,tPen\WObj:=wPaper;
    MoveL Offs(pOrigin,224.5,119.3,0.0),vDraw,z1,tPen\WObj:=wPaper;
    MoveL Offs(pOrigin,224.5,120.1,0.0),vDraw,z1,tPen\WObj:=wPaper;
    MoveL Offs(pOrigin,224.2,120.4,0.0),vDraw,z1,tPen\WObj:=wPaper;
    MoveL Offs(pOrigin,224.2,121.2,0.0),vDraw,z1,tPen\WObj:=wPaper;
    MoveL Offs(pOrigin,223.7,122.0,0.0),vDraw,z1,tPen\WObj:=wPaper;
    MoveL Offs(pOrigin,223.7,122.5,0.0),vDraw,z1,tPen\WObj:=wPaper;
    MoveL Offs(pOrigin,223.4,122.8,0.0),vDraw,z1,tPen\WObj:=wPaper;
    MoveL Offs(pOrigin,222.9,124.1,0.0),vDraw,z1,tPen\WObj:=wPaper;
    MoveL Offs(pOrigin,222.3,124.7,0.0),vDraw,z1,tPen\WObj:=wPaper;
    MoveL Offs(pOrigin,222.1,125.5,0.0),vDraw,z1,tPen\WObj:=wPaper;
    MoveL Offs(pOrigin,221.5,126.0,0.0),vDraw,z1,tPen\WObj:=wPaper;
    MoveL Offs(pOrigin,221.5,126.3,0.0),vDraw,z1,tPen\WObj:=wPaper;
    MoveL Offs(pOrigin,218.3,129.5,0.0),vDraw,z1,tPen\WObj:=wPaper;
    MoveL Offs(pOrigin,218.1,129.5,0.0),vDraw,z1,tPen\WObj:=wPaper;
    MoveL Offs(pOrigin,216.5,130.8,0.0),vDraw,z1,tPen\WObj:=wPaper;
    MoveL Offs(pOrigin,216.2,130.8,0.0),vDraw,z1,tPen\WObj:=wPaper;
    MoveL Offs(pOrigin,213.8,132.1,0.0),vDraw,z1,tPen\WObj:=wPaper;
    MoveL Offs(pOrigin,213.3,132.1,0.0),vDraw,z1,tPen\WObj:=wPaper;
    MoveL Offs(pOrigin,213.0,132.4,0.0),vDraw,z1,tPen\WObj:=wPaper;
    MoveL Offs(pOrigin,212.2,132.4,0.0),vDraw,z1,tPen\WObj:=wPaper;
    MoveL Offs(pOrigin,211.9,132.7,0.0),vDraw,z1,tPen\WObj:=wPaper;
    MoveL Offs(pOrigin,210.9,132.7,0.0),vDraw,z1,tPen\WObj:=wPaper;
    MoveL Offs(pOrigin,210.6,132.9,0.0),vDraw,z1,tPen\WObj:=wPaper;
    MoveL Offs(pOrigin,209.0,132.9,0.0),vDraw,z1,tPen\WObj:=wPaper;
    MoveL Offs(pOrigin,208.7,133.2,0.0),vDraw,z1,tPen\WObj:=wPaper;
    MoveL Offs(pOrigin,202.3,133.2,0.0),vDraw,z1,tPen\WObj:=wPaper;
    MoveL Offs(pOrigin,202.1,132.9,0.0),vDraw,z1,tPen\WObj:=wPaper;
    MoveL Offs(pOrigin,202.1,93.2,0.0),vDraw,fine,tPen\WObj:=wPaper;
    MoveL Offs(pOrigin,202.1,93.2,15.0),vApproach,z5,tPen\WObj:=wPaper;
    MoveL Offs(pOrigin,202.9,90.5,15.0),vTravel,z5,tPen\WObj:=wPaper;
    MoveL Offs(pOrigin,202.9,90.5,0.0),vApproach,fine,tPen\WObj:=wPaper;
    MoveL Offs(pOrigin,202.6,90.3,0.0),vDraw,z1,tPen\WObj:=wPaper;
    MoveL Offs(pOrigin,202.1,90.3,0.0),vDraw,z1,tPen\WObj:=wPaper;
    MoveL Offs(pOrigin,202.1,51.1,0.0),vDraw,z1,tPen\WObj:=wPaper;
    MoveL Offs(pOrigin,202.3,50.8,0.0),vDraw,z1,tPen\WObj:=wPaper;
    MoveL Offs(pOrigin,208.7,50.8,0.0),vDraw,z1,tPen\WObj:=wPaper;
    MoveL Offs(pOrigin,209.0,51.1,0.0),vDraw,z1,tPen\WObj:=wPaper;
    MoveL Offs(pOrigin,210.6,51.1,0.0),vDraw,z1,tPen\WObj:=wPaper;
    MoveL Offs(pOrigin,210.9,51.3,0.0),vDraw,z1,tPen\WObj:=wPaper;
    MoveL Offs(pOrigin,211.9,51.3,0.0),vDraw,z1,tPen\WObj:=wPaper;
    MoveL Offs(pOrigin,212.2,51.6,0.0),vDraw,z1,tPen\WObj:=wPaper;
    MoveL Offs(pOrigin,212.7,51.6,0.0),vDraw,z1,tPen\WObj:=wPaper;
    MoveL Offs(pOrigin,213.0,51.9,0.0),vDraw,z1,tPen\WObj:=wPaper;
    MoveL Offs(pOrigin,213.8,51.9,0.0),vDraw,z1,tPen\WObj:=wPaper;
    MoveL Offs(pOrigin,214.1,52.1,0.0),vDraw,z1,tPen\WObj:=wPaper;
    MoveL Offs(pOrigin,214.6,52.1,0.0),vDraw,z1,tPen\WObj:=wPaper;
    MoveL Offs(pOrigin,215.4,52.7,0.0),vDraw,z1,tPen\WObj:=wPaper;
    MoveL Offs(pOrigin,216.2,52.7,0.0),vDraw,z1,tPen\WObj:=wPaper;
    MoveL Offs(pOrigin,216.5,52.9,0.0),vDraw,z1,tPen\WObj:=wPaper;
    MoveL Offs(pOrigin,216.7,52.9,0.0),vDraw,z1,tPen\WObj:=wPaper;
    MoveL Offs(pOrigin,217.0,53.2,0.0),vDraw,z1,tPen\WObj:=wPaper;
    MoveL Offs(pOrigin,218.9,54.0,0.0),vDraw,z1,tPen\WObj:=wPaper;
    MoveL Offs(pOrigin,219.4,54.5,0.0),vDraw,z1,tPen\WObj:=wPaper;
    MoveL Offs(pOrigin,220.2,54.8,0.0),vDraw,z1,tPen\WObj:=wPaper;
    MoveL Offs(pOrigin,220.7,55.3,0.0),vDraw,z1,tPen\WObj:=wPaper;
    MoveL Offs(pOrigin,221.0,55.3,0.0),vDraw,z1,tPen\WObj:=wPaper;
    MoveL Offs(pOrigin,221.5,55.9,0.0),vDraw,z1,tPen\WObj:=wPaper;
    MoveL Offs(pOrigin,221.8,55.9,0.0),vDraw,z1,tPen\WObj:=wPaper;
    MoveL Offs(pOrigin,223.1,57.2,0.0),vDraw,z1,tPen\WObj:=wPaper;
    MoveL Offs(pOrigin,223.4,57.2,0.0),vDraw,z1,tPen\WObj:=wPaper;
    MoveL Offs(pOrigin,226.1,59.9,0.0),vDraw,z1,tPen\WObj:=wPaper;
    MoveL Offs(pOrigin,226.1,60.1,0.0),vDraw,z1,tPen\WObj:=wPaper;
    MoveL Offs(pOrigin,227.1,61.2,0.0),vDraw,z1,tPen\WObj:=wPaper;
    MoveL Offs(pOrigin,227.1,61.5,0.0),vDraw,z1,tPen\WObj:=wPaper;
    MoveL Offs(pOrigin,228.7,63.6,0.0),vDraw,z1,tPen\WObj:=wPaper;
    MoveL Offs(pOrigin,228.7,63.9,0.0),vDraw,z1,tPen\WObj:=wPaper;
    MoveL Offs(pOrigin,230.3,66.8,0.0),vDraw,z1,tPen\WObj:=wPaper;
    MoveL Offs(pOrigin,230.3,67.3,0.0),vDraw,z1,tPen\WObj:=wPaper;
    MoveL Offs(pOrigin,230.6,67.6,0.0),vDraw,z1,tPen\WObj:=wPaper;
    MoveL Offs(pOrigin,230.6,68.1,0.0),vDraw,z1,tPen\WObj:=wPaper;
    MoveL Offs(pOrigin,230.9,68.4,0.0),vDraw,z1,tPen\WObj:=wPaper;
    MoveL Offs(pOrigin,230.9,68.9,0.0),vDraw,z1,tPen\WObj:=wPaper;
    MoveL Offs(pOrigin,231.1,69.2,0.0),vDraw,z1,tPen\WObj:=wPaper;
    MoveL Offs(pOrigin,231.1,70.0,0.0),vDraw,z1,tPen\WObj:=wPaper;
    MoveL Offs(pOrigin,231.4,70.3,0.0),vDraw,z1,tPen\WObj:=wPaper;
    MoveL Offs(pOrigin,231.4,71.1,0.0),vDraw,z1,tPen\WObj:=wPaper;
    MoveL Offs(pOrigin,231.7,71.3,0.0),vDraw,z1,tPen\WObj:=wPaper;
    MoveL Offs(pOrigin,231.7,72.1,0.0),vDraw,z1,tPen\WObj:=wPaper;
    MoveL Offs(pOrigin,231.9,72.4,0.0),vDraw,z1,tPen\WObj:=wPaper;
    MoveL Offs(pOrigin,231.9,73.7,0.0),vDraw,z1,tPen\WObj:=wPaper;
    MoveL Offs(pOrigin,232.2,74.0,0.0),vDraw,z1,tPen\WObj:=wPaper;
    MoveL Offs(pOrigin,232.2,81.2,0.0),vDraw,z1,tPen\WObj:=wPaper;
    MoveL Offs(pOrigin,231.9,81.5,0.0),vDraw,z1,tPen\WObj:=wPaper;
    MoveL Offs(pOrigin,231.9,82.5,0.0),vDraw,z1,tPen\WObj:=wPaper;
    MoveL Offs(pOrigin,231.7,82.8,0.0),vDraw,z1,tPen\WObj:=wPaper;
  ENDPROC

  PROC Part8()
    MoveL Offs(pOrigin,231.7,83.9,0.0),vDraw,z1,tPen\WObj:=wPaper;
    MoveL Offs(pOrigin,231.4,84.1,0.0),vDraw,z1,tPen\WObj:=wPaper;
    MoveL Offs(pOrigin,231.4,84.9,0.0),vDraw,z1,tPen\WObj:=wPaper;
    MoveL Offs(pOrigin,231.1,85.2,0.0),vDraw,z1,tPen\WObj:=wPaper;
    MoveL Offs(pOrigin,231.1,86.0,0.0),vDraw,z1,tPen\WObj:=wPaper;
    MoveL Offs(pOrigin,230.6,86.8,0.0),vDraw,z1,tPen\WObj:=wPaper;
    MoveL Offs(pOrigin,230.6,87.3,0.0),vDraw,z1,tPen\WObj:=wPaper;
    MoveL Offs(pOrigin,230.3,87.6,0.0),vDraw,z1,tPen\WObj:=wPaper;
    MoveL Offs(pOrigin,230.3,87.9,0.0),vDraw,z1,tPen\WObj:=wPaper;
    MoveL Offs(pOrigin,230.1,88.1,0.0),vDraw,z1,tPen\WObj:=wPaper;
    MoveL Offs(pOrigin,229.3,90.0,0.0),vDraw,z1,tPen\WObj:=wPaper;
    MoveL Offs(pOrigin,228.7,90.5,0.0),vDraw,z1,tPen\WObj:=wPaper;
    MoveL Offs(pOrigin,217.3,90.5,0.0),vDraw,z1,tPen\WObj:=wPaper;
    MoveL Offs(pOrigin,217.0,90.3,0.0),vDraw,z1,tPen\WObj:=wPaper;
    MoveL Offs(pOrigin,216.7,90.5,0.0),vDraw,z1,tPen\WObj:=wPaper;
    MoveL Offs(pOrigin,202.9,90.5,0.0),vDraw,fine,tPen\WObj:=wPaper;
    MoveL Offs(pOrigin,202.9,90.5,15.0),vApproach,z5,tPen\WObj:=wPaper;
  ENDPROC

ENDMODULE
